// TIA Portal V21 export
FUNCTION "GestAzionamentoFesto_CMMT-ST" : Void   // FC43, LAD
{ S7_Optimized_Access := 'TRUE' }
// stored: SetENOAutomatically false
   VAR_INPUT
      "K_AzionamentoFesto_CMMT-ST" : Int;
      K_Motore : Int;
   END_VAR
   VAR_TEMP
      AzionamentoAbilitato : Bool;
      tempDWord : DWord;
      tmpSendBuffer : Array[0..11] of Word;
      tmpReadBuffer : Array[0..11] of Word;
      CambioPosPLC : Bool;
      CambioStatoMotore : Bool;
      ModePosDifferente : Bool;
      CambioStatoEnAxis : Bool;
      ResetRichiesto : Bool;
   END_VAR
   VAR CONSTANT
      MaxCounterStart : Int := 50;
      MAXMODE : Int := 8;
      STATUS_IN_OPERATION : Word := 16#7002;
      ERROR_INVALID_MODE : Word := 16#8202;
      ERROR_OVERRIDE : Word := 16#8203;
      ERROR_INVALID_TRV_BLOCK : Word := 16#8204;
      ERROR_DRIVE_ERROR : Word := 16#8401;
      ERROR_SWITCH_ON_INHIBITED : Word := 16#8402;
      ERROR_DPRD_DAT : Word := 16#8600;
      ERROR_DPWR_DAT : Word := 16#8601;
      Automode : Int := 2;
      JogMode : Int := 7;
      Homing : Int := 4;
   END_VAR
   VAR_TEMP   // added for the SCL form of the ladder/FBD networks
      _w1 : Bool;
   END_VAR
BEGIN

REGION Network 1
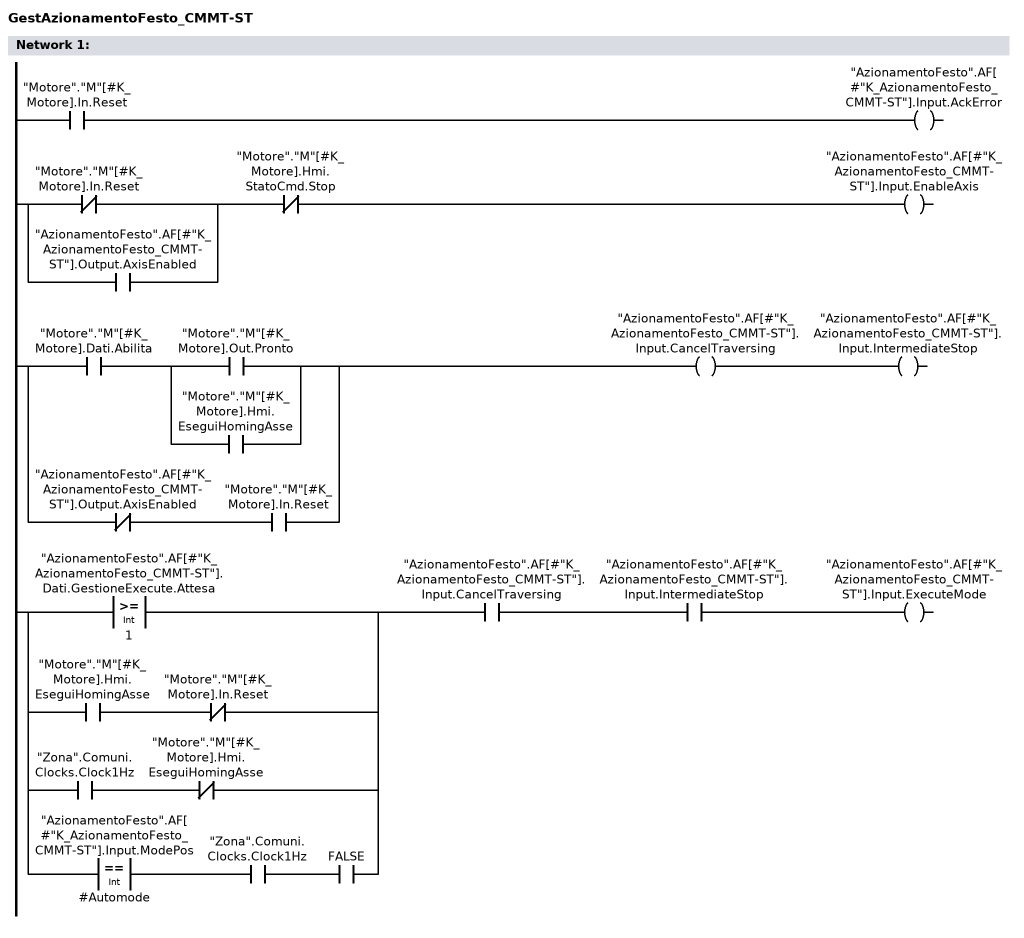
   RUNG wire#powerrail
      Contact( "Motore"."M"[#K_Motore].In.Reset )
      Coil( "AzionamentoFesto".AF[#"K_AzionamentoFesto_CMMT-ST"].Input.AckError )
   END_RUNG
   RUNG wire#powerrail
      I_Contact( "Motore"."M"[#K_Motore].In.Reset )
      wire#w1
      I_Contact( "Motore"."M"[#K_Motore].Hmi.StatoCmd.Stop )
      Coil( "AzionamentoFesto".AF[#"K_AzionamentoFesto_CMMT-ST"].Input.EnableAxis )
   END_RUNG
   RUNG wire#powerrail
      Contact( "AzionamentoFesto".AF[#"K_AzionamentoFesto_CMMT-ST"].Output.AxisEnabled )
   END_RUNG wire#w1
   RUNG wire#powerrail
      Contact( "Motore"."M"[#K_Motore].Dati.Abilita )
      wire#w2
      Contact( "Motore"."M"[#K_Motore].Out.Pronto )
      wire#w3
      Coil( "AzionamentoFesto".AF[#"K_AzionamentoFesto_CMMT-ST"].Input.CancelTraversing )
      Coil( "AzionamentoFesto".AF[#"K_AzionamentoFesto_CMMT-ST"].Input.IntermediateStop )
   END_RUNG
   RUNG wire#w2
      Contact( "Motore"."M"[#K_Motore].Hmi.EseguiHomingAsse )
   END_RUNG wire#w3
   RUNG wire#powerrail
      I_Contact( "AzionamentoFesto".AF[#"K_AzionamentoFesto_CMMT-ST"].Output.AxisEnabled )
      Contact( "Motore"."M"[#K_Motore].In.Reset )
   END_RUNG wire#w3
   RUNG wire#powerrail
      { S7_Templates := "SrcType := Int" } GE_Contact(in1 := "AzionamentoFesto".AF[#"K_AzionamentoFesto_CMMT-ST"].Dati.GestioneExecute.Attesa, in2 := 1)
      wire#w4
      Contact( "AzionamentoFesto".AF[#"K_AzionamentoFesto_CMMT-ST"].Input.CancelTraversing )
      Contact( "AzionamentoFesto".AF[#"K_AzionamentoFesto_CMMT-ST"].Input.IntermediateStop )
      Coil( "AzionamentoFesto".AF[#"K_AzionamentoFesto_CMMT-ST"].Input.ExecuteMode )
   END_RUNG
   RUNG wire#powerrail
      Contact( "Motore"."M"[#K_Motore].Hmi.EseguiHomingAsse )
      I_Contact( "Motore"."M"[#K_Motore].In.Reset )
   END_RUNG wire#w4
   RUNG wire#powerrail
      Contact( "Zona".Comuni.Clocks.Clock1Hz )
      I_Contact( "Motore"."M"[#K_Motore].Hmi.EseguiHomingAsse )
   END_RUNG wire#w4
   RUNG wire#powerrail
      { S7_Templates := "SrcType := Int" } EQ_Contact(in1 := "AzionamentoFesto".AF[#"K_AzionamentoFesto_CMMT-ST"].Input.ModePos, in2 := #Automode)
      Contact( "Zona".Comuni.Clocks.Clock1Hz )
      Contact( FALSE )
   END_RUNG wire#w4
   // the same network as SCL:
   "AzionamentoFesto".AF[#"K_AzionamentoFesto_CMMT-ST"].Input.AckError := "Motore"."M"[#K_Motore].In.Reset;
   "AzionamentoFesto".AF[#"K_AzionamentoFesto_CMMT-ST"].Input.EnableAxis := (NOT "Motore"."M"[#K_Motore].In.Reset OR "AzionamentoFesto".AF[#"K_AzionamentoFesto_CMMT-ST"].Output.AxisEnabled) AND NOT "Motore"."M"[#K_Motore].Hmi.StatoCmd.Stop;
   #_w1 := ("Motore"."M"[#K_Motore].Dati.Abilita AND ("Motore"."M"[#K_Motore].Out.Pronto OR "Motore"."M"[#K_Motore].Hmi.EseguiHomingAsse)) OR (NOT "AzionamentoFesto".AF[#"K_AzionamentoFesto_CMMT-ST"].Output.AxisEnabled AND "Motore"."M"[#K_Motore].In.Reset);
   "AzionamentoFesto".AF[#"K_AzionamentoFesto_CMMT-ST"].Input.CancelTraversing := #_w1;
   "AzionamentoFesto".AF[#"K_AzionamentoFesto_CMMT-ST"].Input.IntermediateStop := #_w1;
   "AzionamentoFesto".AF[#"K_AzionamentoFesto_CMMT-ST"].Input.ExecuteMode := (("AzionamentoFesto".AF[#"K_AzionamentoFesto_CMMT-ST"].Dati.GestioneExecute.Attesa >= 1) OR ("Motore"."M"[#K_Motore].Hmi.EseguiHomingAsse AND NOT "Motore"."M"[#K_Motore].In.Reset) OR ("Zona".Comuni.Clocks.Clock1Hz AND NOT "Motore"."M"[#K_Motore].Hmi.EseguiHomingAsse) OR (("AzionamentoFesto".AF[#"K_AzionamentoFesto_CMMT-ST"].Input.ModePos = #Automode) AND "Zona".Comuni.Clocks.Clock1Hz AND FALSE)) AND "AzionamentoFesto".AF[#"K_AzionamentoFesto_CMMT-ST"].Input.CancelTraversing AND "AzionamentoFesto".AF[#"K_AzionamentoFesto_CMMT-ST"].Input.IntermediateStop;
END_REGION

REGION Network 2 (SCL)
   REGION Modifiche from BRAIN ELECTRIC     

       "AzionamentoFesto".AF[#"K_AzionamentoFesto_CMMT-ST"].Input.HardwareId := "Motore".M[#K_Motore].In.ProfinetHwSubModule;
       "AzionamentoFesto".AF[#"K_AzionamentoFesto_CMMT-ST"].Input.Position := REAL_TO_DINT("Motore".M[#K_Motore].In.CmdPosizioneRich);
       "AzionamentoFesto".AF[#"K_AzionamentoFesto_CMMT-ST"].Input.Velocity := REAL_TO_INT("Motore".M[#K_Motore].In.CmdVelocitaRich);
       "AzionamentoFesto".AF[#"K_AzionamentoFesto_CMMT-ST"].Input.ConfigEPos := 15;



       REGION Comando execute nel motore

           IF "AzionamentoFesto".AF[#"K_AzionamentoFesto_CMMT-ST"].Dati.GestioneExecute.Richiesto AND "AzionamentoFesto".AF[#"K_AzionamentoFesto_CMMT-ST"].Dati.GestioneExecute.Attesa <= 5 THEN
               "AzionamentoFesto".AF[#"K_AzionamentoFesto_CMMT-ST"].Dati.GestioneExecute.Attesa += 1;
           END_IF;
           IF "AzionamentoFesto".AF[#"K_AzionamentoFesto_CMMT-ST"].Dati.GestioneExecute.Attesa >= 1 THEN
               "AzionamentoFesto".AF[#"K_AzionamentoFesto_CMMT-ST"].Dati.GestioneExecute.Durata += 1;
           END_IF;
           IF "AzionamentoFesto".AF[#"K_AzionamentoFesto_CMMT-ST"].Dati.GestioneExecute.Durata >= 2 OR "Motore".M[#K_Motore].Hmi.EseguiHomingAsse THEN
               "AzionamentoFesto".AF[#"K_AzionamentoFesto_CMMT-ST"].Dati.GestioneExecute.Richiesto := False;
               "AzionamentoFesto".AF[#"K_AzionamentoFesto_CMMT-ST"].Dati.GestioneExecute.Attesa :=
               "AzionamentoFesto".AF[#"K_AzionamentoFesto_CMMT-ST"].Dati.GestioneExecute.Durata := 0;
           END_IF;

               #CambioPosPLC := "AzionamentoFesto".AF[#"K_AzionamentoFesto_CMMT-ST"].Dati.GestioneExecute.OldPosition <> "AzionamentoFesto".AF[#"K_AzionamentoFesto_CMMT-ST"].Input.Position;
               #CambioStatoMotore := "AzionamentoFesto".AF[#"K_AzionamentoFesto_CMMT-ST"].Dati.GestioneExecute.OldStatoMotore <> "Motore".M[#K_Motore].Hmi.StatoMotore;
               #ModePosDifferente := "AzionamentoFesto".AF[#"K_AzionamentoFesto_CMMT-ST"].Input.ModePos <> "AzionamentoFesto".AF[#"K_AzionamentoFesto_CMMT-ST"].Dati.GestioneExecute.OldModePos;
               #CambioStatoEnAxis := "AzionamentoFesto".AF[#"K_AzionamentoFesto_CMMT-ST"].Input.EnableAxis <> "AzionamentoFesto".AF[#"K_AzionamentoFesto_CMMT-ST"].Dati.GestioneExecute.OldAxisEnable;
               #ResetRichiesto := "Motore".M[#K_Motore].In.Reset <> "AzionamentoFesto".AF[#"K_AzionamentoFesto_CMMT-ST"].Dati.GestioneExecute.OldResetState;
               IF #CambioPosPLC OR #CambioStatoMotore OR #ModePosDifferente OR #CambioStatoEnAxis OR #ResetRichiesto THEN
                   "AzionamentoFesto".AF[#"K_AzionamentoFesto_CMMT-ST"].Dati.GestioneExecute.OldPosition := "AzionamentoFesto".AF[#"K_AzionamentoFesto_CMMT-ST"].Input.Position;
                   "AzionamentoFesto".AF[#"K_AzionamentoFesto_CMMT-ST"].Dati.GestioneExecute.OldStatoMotore := "Motore".M[#K_Motore].Hmi.StatoMotore;
                   "AzionamentoFesto".AF[#"K_AzionamentoFesto_CMMT-ST"].Dati.GestioneExecute.OldAxisEnable := "AzionamentoFesto".AF[#"K_AzionamentoFesto_CMMT-ST"].Input.EnableAxis;
                   "AzionamentoFesto".AF[#"K_AzionamentoFesto_CMMT-ST"].Dati.GestioneExecute.OldModePos := "AzionamentoFesto".AF[#"K_AzionamentoFesto_CMMT-ST"].Input.ModePos;
                   "AzionamentoFesto".AF[#"K_AzionamentoFesto_CMMT-ST"].Dati.GestioneExecute.OldResetState := "Motore".M[#K_Motore].In.Reset;
                   "AzionamentoFesto".AF[#"K_AzionamentoFesto_CMMT-ST"].Dati.GestioneExecute.Richiesto := True;
               END_IF;
           END_REGION ;


       IF "Zona".Comuni.FirstScanFromCpu OR NOT "AzionamentoFesto".AF[#"K_AzionamentoFesto_CMMT-ST"].Output.AxisRef THEN
           "Motore".M[#K_Motore].Allarmi.A[KAllMot_RichiestaAzzeramento].Stato := True;
       END_IF;

       "Motore".M[#K_Motore].Out.PosAttuale := "AzionamentoFesto".AF[#"K_AzionamentoFesto_CMMT-ST"].Output.ActPosition;
       "Motore".M[#K_Motore].Allarmi.A[KAllMot_DriveInAllarme].Stato := "AzionamentoFesto".AF[#"K_AzionamentoFesto_CMMT-ST"].Output.AxisError;
       #AzionamentoAbilitato := "AzionamentoFesto".AF[#"K_AzionamentoFesto_CMMT-ST"].Output.AxisEnabled;

       IF NOT "Motore".M[#K_Motore].Hmi.EseguiHomingAsse THEN
           IF "Motore".M[#K_Motore].Hmi.StatoCmd.Stop OR NOT #AzionamentoAbilitato THEN
               "AzionamentoFesto".AF[#"K_AzionamentoFesto_CMMT-ST"].Input.ModePos := #Automode;
               "AzionamentoFesto".AF[#"K_AzionamentoFesto_CMMT-ST"].Input.Jog1 := False;
               "AzionamentoFesto".AF[#"K_AzionamentoFesto_CMMT-ST"].Input.Jog2 := False;
               "AzionamentoFesto".AF[#"K_AzionamentoFesto_CMMT-ST"].Input.OverV := 0;
               "AzionamentoFesto".AF[#"K_AzionamentoFesto_CMMT-ST"].Input.Velocity := 0;
           ELSIF "Motore".M[#K_Motore].Hmi.StatoCmd.Auto THEN
               "AzionamentoFesto".AF[#"K_AzionamentoFesto_CMMT-ST"].Input.ModePos := #Automode;
               "AzionamentoFesto".AF[#"K_AzionamentoFesto_CMMT-ST"].Input.Jog1 := False;
               "AzionamentoFesto".AF[#"K_AzionamentoFesto_CMMT-ST"].Input.Jog2 := False;
               "AzionamentoFesto".AF[#"K_AzionamentoFesto_CMMT-ST"].Input.OverV := 100;
           ELSIF "Motore".M[#K_Motore].Hmi.StatoCmd.ManPos THEN
               "AzionamentoFesto".AF[#"K_AzionamentoFesto_CMMT-ST"].Input.ModePos := #JogMode;
               "AzionamentoFesto".AF[#"K_AzionamentoFesto_CMMT-ST"].Input.Jog1 := True;
               "AzionamentoFesto".AF[#"K_AzionamentoFesto_CMMT-ST"].Input.OverV := REAL_TO_INT("Motore".M[#K_Motore].Hmi.VelManuale);
           ELSIF "Motore".M[#K_Motore].Hmi.StatoCmd.ManNeg THEN
               "AzionamentoFesto".AF[#"K_AzionamentoFesto_CMMT-ST"].Input.ModePos := #JogMode;
               "AzionamentoFesto".AF[#"K_AzionamentoFesto_CMMT-ST"].Input.Jog2 := True;
               "AzionamentoFesto".AF[#"K_AzionamentoFesto_CMMT-ST"].Input.OverV := REAL_TO_INT("Motore".M[#K_Motore].Hmi.VelManuale);
           END_IF;
       ELSE
           "AzionamentoFesto".AF[#"K_AzionamentoFesto_CMMT-ST"].Input.ModePos := #Homing;
           "AzionamentoFesto".AF[#"K_AzionamentoFesto_CMMT-ST"].Input.Jog1 := False;
           "AzionamentoFesto".AF[#"K_AzionamentoFesto_CMMT-ST"].Input.Jog2 := False;
           "AzionamentoFesto".AF[#"K_AzionamentoFesto_CMMT-ST"].Input.OverV := REAL_TO_INT("Motore".M[#K_Motore].Hmi.VelManuale);
           "AzionamentoFesto".AF[#"K_AzionamentoFesto_CMMT-ST"].Input.Velocity := 100;
       END_IF;
       IF "AzionamentoFesto".AF[#"K_AzionamentoFesto_CMMT-ST"].Output.AxisRef AND "Motore".M[#K_Motore].Hmi.EseguiHomingAsse THEN //OR NOT "AzionamentiFesto".AF[#"K_AzionamentoFesto_CMMT-ST"].Input.EnableAxis THEN
           "Motore".M[#K_Motore].Hmi.EseguiHomingAsse := False;
           "Motore".M[#K_Motore].Allarmi.A[KAllMot_RichiestaAzzeramento].Stato := False;
       END_IF;

   END_REGION
   REGION Check OPM and Override Values
       // Check the Mode of Operation
       IF "AzionamentoFesto".AF[#"K_AzionamentoFesto_CMMT-ST"].Input.ModePos > #MAXMODE THEN
           "AzionamentoFesto".AF[#"K_AzionamentoFesto_CMMT-ST"].Output.Error := True;
           "AzionamentoFesto".AF[#"K_AzionamentoFesto_CMMT-ST"].Dati.Status := #ERROR_INVALID_MODE;
           "AzionamentoFesto".AF[#"K_AzionamentoFesto_CMMT-ST"].Dati.ExecuteIntern := false;
       ELSIF "AzionamentoFesto".AF[#"K_AzionamentoFesto_CMMT-ST"].Input.ModePos < 1 THEN
           "AzionamentoFesto".AF[#"K_AzionamentoFesto_CMMT-ST"].Output.Error := True;
           "AzionamentoFesto".AF[#"K_AzionamentoFesto_CMMT-ST"].Dati.Status := #ERROR_INVALID_MODE;
           "AzionamentoFesto".AF[#"K_AzionamentoFesto_CMMT-ST"].Dati.ExecuteIntern := false;
       ELSE
           IF "AzionamentoFesto".AF[#"K_AzionamentoFesto_CMMT-ST"].Dati.Status = #ERROR_INVALID_MODE THEN
               "AzionamentoFesto".AF[#"K_AzionamentoFesto_CMMT-ST"].Dati.Status := #STATUS_IN_OPERATION;
               "AzionamentoFesto".AF[#"K_AzionamentoFesto_CMMT-ST"].Output.Error := False;
           END_IF;
       END_IF;


       //Check the Velocity Override 
       IF ("AzionamentoFesto".AF[#"K_AzionamentoFesto_CMMT-ST"].Input.OverV < 0) OR ("AzionamentoFesto".AF[#"K_AzionamentoFesto_CMMT-ST"].Input.OverV > 199) THEN
           "AzionamentoFesto".AF[#"K_AzionamentoFesto_CMMT-ST"].Dati.Status := #ERROR_OVERRIDE;
           "AzionamentoFesto".AF[#"K_AzionamentoFesto_CMMT-ST"].Output.Error := True;
       ELSE
           // Write Velocity Override into Send Buffer
           "AzionamentoFesto".AF[#"K_AzionamentoFesto_CMMT-ST"].Dati.CycWrite.Override := INT_TO_WORD(REAL_TO_INT(16384.0 * (INT_TO_REAL("AzionamentoFesto".AF[#"K_AzionamentoFesto_CMMT-ST"].Input.OverV) / 100.0)));
           IF "AzionamentoFesto".AF[#"K_AzionamentoFesto_CMMT-ST"].Dati.Status = #ERROR_OVERRIDE THEN
               "AzionamentoFesto".AF[#"K_AzionamentoFesto_CMMT-ST"].Dati.Status := #STATUS_IN_OPERATION;
               "AzionamentoFesto".AF[#"K_AzionamentoFesto_CMMT-ST"].Output.Error := False;
           END_IF;
       END_IF;

       //Check the Acceleration Override  (0% - 100%, 100% => W#16#4000)
       IF ("AzionamentoFesto".AF[#"K_AzionamentoFesto_CMMT-ST"].Input.OverAcc < 0) OR ("AzionamentoFesto".AF[#"K_AzionamentoFesto_CMMT-ST"].Input.OverAcc > 100) THEN
           "AzionamentoFesto".AF[#"K_AzionamentoFesto_CMMT-ST"].Dati.Status := #ERROR_OVERRIDE;
           "AzionamentoFesto".AF[#"K_AzionamentoFesto_CMMT-ST"].Output.Error := True;
       ELSE
           // Write Acceleration Override into Send Buffer
           "AzionamentoFesto".AF[#"K_AzionamentoFesto_CMMT-ST"].Dati.CycWrite.MDI_ACC := INT_TO_WORD(REAL_TO_INT(16384.0 * (INT_TO_REAL("AzionamentoFesto".AF[#"K_AzionamentoFesto_CMMT-ST"].Input.OverAcc) / 100.0)));
           IF "AzionamentoFesto".AF[#"K_AzionamentoFesto_CMMT-ST"].Dati.Status = #ERROR_OVERRIDE THEN
               "AzionamentoFesto".AF[#"K_AzionamentoFesto_CMMT-ST"].Dati.Status := #STATUS_IN_OPERATION;
               "AzionamentoFesto".AF[#"K_AzionamentoFesto_CMMT-ST"].Output.Error := False;
           END_IF;
       END_IF;

       //Check the Deceleration Override  (0% - 100%, 100% => W#16#4000)
       IF ("AzionamentoFesto".AF[#"K_AzionamentoFesto_CMMT-ST"].Input.OverDec < 0) OR ("AzionamentoFesto".AF[#"K_AzionamentoFesto_CMMT-ST"].Input.OverDec > 100) THEN
           "AzionamentoFesto".AF[#"K_AzionamentoFesto_CMMT-ST"].Dati.Status := #ERROR_OVERRIDE;
           "AzionamentoFesto".AF[#"K_AzionamentoFesto_CMMT-ST"].Output.Error := True;
       ELSE
           // Write Deceleration Override into Send Buffer
           "AzionamentoFesto".AF[#"K_AzionamentoFesto_CMMT-ST"].Dati.CycWrite.MDI_DEC := INT_TO_WORD(REAL_TO_INT(16384.0 * (INT_TO_REAL("AzionamentoFesto".AF[#"K_AzionamentoFesto_CMMT-ST"].Input.OverDec) / 100.0)));
           IF "AzionamentoFesto".AF[#"K_AzionamentoFesto_CMMT-ST"].Dati.Status = #ERROR_OVERRIDE THEN
               "AzionamentoFesto".AF[#"K_AzionamentoFesto_CMMT-ST"].Dati.Status := #STATUS_IN_OPERATION;
               "AzionamentoFesto".AF[#"K_AzionamentoFesto_CMMT-ST"].Output.Error := False;
           END_IF;
       END_IF;
   END_REGION ;

   REGION Lettura della status word
       // Read cyclic telegram 111
       "AzionamentoFesto".AF[#"K_AzionamentoFesto_CMMT-ST"].Dati.RetDPRD := DPRD_DAT(LADDR := "AzionamentoFesto".AF[#"K_AzionamentoFesto_CMMT-ST"].Input.HardwareId,
                                                                                     RECORD => #tmpReadBuffer);

       //check if the return code is unequal zero -> error occured
       IF "AzionamentoFesto".AF[#"K_AzionamentoFesto_CMMT-ST"].Dati.RetDPRD <> 0 THEN
           "AzionamentoFesto".AF[#"K_AzionamentoFesto_CMMT-ST"].Output.Error := true;
           "AzionamentoFesto".AF[#"K_AzionamentoFesto_CMMT-ST"].Dati.Status := #ERROR_DPRD_DAT;
           "AzionamentoFesto".AF[#"K_AzionamentoFesto_CMMT-ST"].Output.DiagID := INT_TO_WORD("AzionamentoFesto".AF[#"K_AzionamentoFesto_CMMT-ST"].Dati.RetDPRD);
       ELSE

           // set the Diag status back "in operation"
           IF "AzionamentoFesto".AF[#"K_AzionamentoFesto_CMMT-ST"].Dati.Status = #ERROR_DPRD_DAT THEN
               "AzionamentoFesto".AF[#"K_AzionamentoFesto_CMMT-ST"].Dati.Status := #STATUS_IN_OPERATION;
               "AzionamentoFesto".AF[#"K_AzionamentoFesto_CMMT-ST"].Output.DiagID := 0;
               "AzionamentoFesto".AF[#"K_AzionamentoFesto_CMMT-ST"].Output.Error := False;
           END_IF;
       END_IF;

   END_REGION ;


   REGION Read Input from temp data
       // copy all values from tmp buffer to static data
       // ZSW1
       "AzionamentoFesto".AF[#"K_AzionamentoFesto_CMMT-ST"].Dati.CycRead.ZSW1.followingErrorInTolerance := #tmpReadBuffer[0].%X8;
       "AzionamentoFesto".AF[#"K_AzionamentoFesto_CMMT-ST"].Dati.CycRead.ZSW1.controlRequest := #tmpReadBuffer[0].%X9;
       "AzionamentoFesto".AF[#"K_AzionamentoFesto_CMMT-ST"].Dati.CycRead.ZSW1.targetPosReached := #tmpReadBuffer[0].%X10;
       "AzionamentoFesto".AF[#"K_AzionamentoFesto_CMMT-ST"].Dati.CycRead.ZSW1.homePosSet := #tmpReadBuffer[0].%X11;
       "AzionamentoFesto".AF[#"K_AzionamentoFesto_CMMT-ST"].Dati.CycRead.ZSW1.acknowledgeTraversingBlockActivated := #tmpReadBuffer[0].%X12;
       "AzionamentoFesto".AF[#"K_AzionamentoFesto_CMMT-ST"].Dati.CycRead.ZSW1.driveStopped := #tmpReadBuffer[0].%X13;
       "AzionamentoFesto".AF[#"K_AzionamentoFesto_CMMT-ST"].Dati.CycRead.ZSW1.axisAccelerates := #tmpReadBuffer[0].%X14;
       "AzionamentoFesto".AF[#"K_AzionamentoFesto_CMMT-ST"].Dati.CycRead.ZSW1.axisDecelerates := #tmpReadBuffer[0].%X15;
       "AzionamentoFesto".AF[#"K_AzionamentoFesto_CMMT-ST"].Dati.CycRead.ZSW1.readyForSwitchOn := #tmpReadBuffer[0].%X0;
       "AzionamentoFesto".AF[#"K_AzionamentoFesto_CMMT-ST"].Dati.CycRead.ZSW1.ready := #tmpReadBuffer[0].%X1;
       "AzionamentoFesto".AF[#"K_AzionamentoFesto_CMMT-ST"].Dati.CycRead.ZSW1.operationEnabled := #tmpReadBuffer[0].%X2;
       "AzionamentoFesto".AF[#"K_AzionamentoFesto_CMMT-ST"].Dati.CycRead.ZSW1.faultPresent := #tmpReadBuffer[0].%X3;
       "AzionamentoFesto".AF[#"K_AzionamentoFesto_CMMT-ST"].Dati.CycRead.ZSW1.noCoastingActive := #tmpReadBuffer[0].%X4;
       "AzionamentoFesto".AF[#"K_AzionamentoFesto_CMMT-ST"].Dati.CycRead.ZSW1.noQuickStopActive := #tmpReadBuffer[0].%X5;
       "AzionamentoFesto".AF[#"K_AzionamentoFesto_CMMT-ST"].Dati.CycRead.ZSW1.switchingOnInhibitedActive := #tmpReadBuffer[0].%X6;
       "AzionamentoFesto".AF[#"K_AzionamentoFesto_CMMT-ST"].Dati.CycRead.ZSW1.warningActive := #tmpReadBuffer[0].%X7;

       //POS_ZSW1
       "AzionamentoFesto".AF[#"K_AzionamentoFesto_CMMT-ST"].Dati.CycRead.POS_ZSW1 := #tmpReadBuffer[1];
       "AzionamentoFesto".AF[#"K_AzionamentoFesto_CMMT-ST"].Output.EPosZSW1 := "AzionamentoFesto".AF[#"K_AzionamentoFesto_CMMT-ST"].Dati.CycRead.POS_ZSW1;

       //POS_ZSW2
       "AzionamentoFesto".AF[#"K_AzionamentoFesto_CMMT-ST"].Dati.CycRead.POS_ZSW2 := #tmpReadBuffer[2];
       "AzionamentoFesto".AF[#"K_AzionamentoFesto_CMMT-ST"].Output.EPosZSW2 := "AzionamentoFesto".AF[#"K_AzionamentoFesto_CMMT-ST"].Dati.CycRead.POS_ZSW2;

       // ZSW2
       "AzionamentoFesto".AF[#"K_AzionamentoFesto_CMMT-ST"].Dati.CycRead.ZSW2.deviceSpecificBit8 := #tmpReadBuffer[3].%X8;
       "AzionamentoFesto".AF[#"K_AzionamentoFesto_CMMT-ST"].Dati.CycRead.ZSW2.deviceSpecificBit9 := #tmpReadBuffer[3].%X9;
       "AzionamentoFesto".AF[#"K_AzionamentoFesto_CMMT-ST"].Dati.CycRead.ZSW2.deviceSpecificBit10 := #tmpReadBuffer[3].%X10;
       "AzionamentoFesto".AF[#"K_AzionamentoFesto_CMMT-ST"].Dati.CycRead.ZSW2.deviceSpecificBit11 := #tmpReadBuffer[3].%X11;
       "AzionamentoFesto".AF[#"K_AzionamentoFesto_CMMT-ST"].Dati.CycRead.ZSW2.doSignOfLifeBit0 := #tmpReadBuffer[3].%X12;
       "AzionamentoFesto".AF[#"K_AzionamentoFesto_CMMT-ST"].Dati.CycRead.ZSW2.doSignOfLifeBit1 := #tmpReadBuffer[3].%X13;
       "AzionamentoFesto".AF[#"K_AzionamentoFesto_CMMT-ST"].Dati.CycRead.ZSW2.doSignOfLifeBit2 := #tmpReadBuffer[3].%X14;
       "AzionamentoFesto".AF[#"K_AzionamentoFesto_CMMT-ST"].Dati.CycRead.ZSW2.doSignOfLifeBit3 := #tmpReadBuffer[3].%X15;
       "AzionamentoFesto".AF[#"K_AzionamentoFesto_CMMT-ST"].Dati.CycRead.ZSW2.deviceSpecificBit0 := #tmpReadBuffer[3].%X0;
       "AzionamentoFesto".AF[#"K_AzionamentoFesto_CMMT-ST"].Dati.CycRead.ZSW2.deviceSpecificBit1 := #tmpReadBuffer[3].%X1;
       "AzionamentoFesto".AF[#"K_AzionamentoFesto_CMMT-ST"].Dati.CycRead.ZSW2.deviceSpecificBit2 := #tmpReadBuffer[3].%X2;
       "AzionamentoFesto".AF[#"K_AzionamentoFesto_CMMT-ST"].Dati.CycRead.ZSW2.deviceSpecificBit3 := #tmpReadBuffer[3].%X3;
       "AzionamentoFesto".AF[#"K_AzionamentoFesto_CMMT-ST"].Dati.CycRead.ZSW2.deviceSpecificBit4 := #tmpReadBuffer[3].%X4;
       "AzionamentoFesto".AF[#"K_AzionamentoFesto_CMMT-ST"].Dati.CycRead.ZSW2.deviceSpecificBit5 := #tmpReadBuffer[3].%X5;
       "AzionamentoFesto".AF[#"K_AzionamentoFesto_CMMT-ST"].Dati.CycRead.ZSW2.deviceSpecificBit6 := #tmpReadBuffer[3].%X6;
       "AzionamentoFesto".AF[#"K_AzionamentoFesto_CMMT-ST"].Dati.CycRead.ZSW2.deviceSpecificBit7 := #tmpReadBuffer[3].%X7;

       //MELDW
       "AzionamentoFesto".AF[#"K_AzionamentoFesto_CMMT-ST"].Dati.CycRead.MELDW := #tmpReadBuffer[4];

       //XIST_A
       "AzionamentoFesto".AF[#"K_AzionamentoFesto_CMMT-ST"].Dati.CycRead.XIST_A.%W0 := #tmpReadBuffer[6];
       "AzionamentoFesto".AF[#"K_AzionamentoFesto_CMMT-ST"].Dati.CycRead.XIST_A.%W1 := #tmpReadBuffer[5];

       //NIST_B
       "AzionamentoFesto".AF[#"K_AzionamentoFesto_CMMT-ST"].Dati.CycRead.NIST_B.%W0 := #tmpReadBuffer[8];
       "AzionamentoFesto".AF[#"K_AzionamentoFesto_CMMT-ST"].Dati.CycRead.NIST_B.%W1 := #tmpReadBuffer[7];

       //Fault_Code
       "AzionamentoFesto".AF[#"K_AzionamentoFesto_CMMT-ST"].Dati.CycRead.Fault_Code := #tmpReadBuffer[9];

       //Warn_Code
       "AzionamentoFesto".AF[#"K_AzionamentoFesto_CMMT-ST"].Dati.CycRead.Warn_Code := #tmpReadBuffer[10];

       //Reserved
       "AzionamentoFesto".AF[#"K_AzionamentoFesto_CMMT-ST"].Dati.CycRead.Reserved := #tmpReadBuffer[11];
   END_REGION ;

   // Mapping of the FB Outputs
   "AzionamentoFesto".AF[#"K_AzionamentoFesto_CMMT-ST"].Output.AxisEnabled := "AzionamentoFesto".AF[#"K_AzionamentoFesto_CMMT-ST"].Dati.CycRead.ZSW1.operationEnabled;
   "AzionamentoFesto".AF[#"K_AzionamentoFesto_CMMT-ST"].Output.AxisError := "AzionamentoFesto".AF[#"K_AzionamentoFesto_CMMT-ST"].Dati.CycRead.ZSW1.faultPresent;
   "AzionamentoFesto".AF[#"K_AzionamentoFesto_CMMT-ST"].Output.AxisWarn := "AzionamentoFesto".AF[#"K_AzionamentoFesto_CMMT-ST"].Dati.CycRead.ZSW1.warningActive;
   "AzionamentoFesto".AF[#"K_AzionamentoFesto_CMMT-ST"].Output.AxisPosOk := "AzionamentoFesto".AF[#"K_AzionamentoFesto_CMMT-ST"].Dati.CycRead.ZSW1.targetPosReached;
   "AzionamentoFesto".AF[#"K_AzionamentoFesto_CMMT-ST"].Output.AxisRef := "AzionamentoFesto".AF[#"K_AzionamentoFesto_CMMT-ST"].Dati.CycRead.ZSW1.homePosSet;
   "AzionamentoFesto".AF[#"K_AzionamentoFesto_CMMT-ST"].Output.AxisAckSetpoint := "AzionamentoFesto".AF[#"K_AzionamentoFesto_CMMT-ST"].Dati.CycRead.ZSW1.acknowledgeTraversingBlockActivated;
   "AzionamentoFesto".AF[#"K_AzionamentoFesto_CMMT-ST"].Output.ClampTorqueReached := "AzionamentoFesto".AF[#"K_AzionamentoFesto_CMMT-ST"].Dati.CycRead.POS_ZSW2.%X13;
   "AzionamentoFesto".AF[#"K_AzionamentoFesto_CMMT-ST"].Output.AxisSpFixed := "AzionamentoFesto".AF[#"K_AzionamentoFesto_CMMT-ST"].Dati.CycRead.ZSW1.driveStopped;
   "AzionamentoFesto".AF[#"K_AzionamentoFesto_CMMT-ST"].Output.ActVelocity := "AzionamentoFesto".AF[#"K_AzionamentoFesto_CMMT-ST"].Dati.CycRead.NIST_B;


   //scaling the ActVelocity output
   IF "AzionamentoFesto".AF[#"K_AzionamentoFesto_CMMT-ST"].Input.BaseSpeedValue <> 0 THEN
       "AzionamentoFesto".AF[#"K_AzionamentoFesto_CMMT-ST"].Output.ActVelocity := "AzionamentoFesto".AF[#"K_AzionamentoFesto_CMMT-ST"].Output.ActVelocity * (("AzionamentoFesto".AF[#"K_AzionamentoFesto_CMMT-ST"].Input.BaseSpeedValue / 1073741824.0));
   END_IF;

   "AzionamentoFesto".AF[#"K_AzionamentoFesto_CMMT-ST"].Output.ActPosition := "AzionamentoFesto".AF[#"K_AzionamentoFesto_CMMT-ST"].Dati.CycRead.XIST_A;
   "AzionamentoFesto".AF[#"K_AzionamentoFesto_CMMT-ST"].Output.ActWarn := "AzionamentoFesto".AF[#"K_AzionamentoFesto_CMMT-ST"].Dati.CycRead.Warn_Code;
   "AzionamentoFesto".AF[#"K_AzionamentoFesto_CMMT-ST"].Output.ActFault := "AzionamentoFesto".AF[#"K_AzionamentoFesto_CMMT-ST"].Dati.CycRead.Fault_Code;
   "AzionamentoFesto".AF[#"K_AzionamentoFesto_CMMT-ST"].Output.Lockout := "AzionamentoFesto".AF[#"K_AzionamentoFesto_CMMT-ST"].Dati.CycRead.ZSW1.switchingOnInhibitedActive;

   //Check the drive error and Lockout status
   IF "AzionamentoFesto".AF[#"K_AzionamentoFesto_CMMT-ST"].Output.AxisError THEN
       "AzionamentoFesto".AF[#"K_AzionamentoFesto_CMMT-ST"].Dati.Status := #ERROR_DRIVE_ERROR;
       "AzionamentoFesto".AF[#"K_AzionamentoFesto_CMMT-ST"].Output.Error := True;
   ELSIF "AzionamentoFesto".AF[#"K_AzionamentoFesto_CMMT-ST"].Output.Lockout THEN
       "AzionamentoFesto".AF[#"K_AzionamentoFesto_CMMT-ST"].Dati.Status := #ERROR_SWITCH_ON_INHIBITED;
       "AzionamentoFesto".AF[#"K_AzionamentoFesto_CMMT-ST"].Output.Error := True;
   ELSE
       // error is gone -> set status in operational
       IF ("AzionamentoFesto".AF[#"K_AzionamentoFesto_CMMT-ST"].Dati.Status = #ERROR_DRIVE_ERROR) OR "AzionamentoFesto".AF[#"K_AzionamentoFesto_CMMT-ST"].Dati.Status = #ERROR_SWITCH_ON_INHIBITED THEN
           "AzionamentoFesto".AF[#"K_AzionamentoFesto_CMMT-ST"].Dati.Status := #STATUS_IN_OPERATION;
           "AzionamentoFesto".AF[#"K_AzionamentoFesto_CMMT-ST"].Output.Error := False;
       END_IF;
   END_IF;

   //Enable the Axis
   "AzionamentoFesto".AF[#"K_AzionamentoFesto_CMMT-ST"].Dati.CycWrite.STW1.on := "AzionamentoFesto".AF[#"K_AzionamentoFesto_CMMT-ST"].Input.EnableAxis;                       //STW1.0

   //fix values for STW1 data
   "AzionamentoFesto".AF[#"K_AzionamentoFesto_CMMT-ST"].Dati.CycWrite.STW1.cancelTraversing := "AzionamentoFesto".AF[#"K_AzionamentoFesto_CMMT-ST"].Input.CancelTraversing;   //STW1.4
   "AzionamentoFesto".AF[#"K_AzionamentoFesto_CMMT-ST"].Dati.CycWrite.STW1.intermediateStop := "AzionamentoFesto".AF[#"K_AzionamentoFesto_CMMT-ST"].Input.IntermediateStop;   //STW1.5
   "AzionamentoFesto".AF[#"K_AzionamentoFesto_CMMT-ST"].Dati.CycWrite.STW1.acknowledgeFault := "AzionamentoFesto".AF[#"K_AzionamentoFesto_CMMT-ST"].Input.AckError;           //STW1.7
   "AzionamentoFesto".AF[#"K_AzionamentoFesto_CMMT-ST"].Dati.CycWrite.STW1.controlByPlc := TRUE;                    //STW1.10
   "AzionamentoFesto".AF[#"K_AzionamentoFesto_CMMT-ST"].Dati.CycWrite.STW1.enableOperation := TRUE;                 //STW1.3

   // copy the position set value into the send struct
   IF "AzionamentoFesto".AF[#"K_AzionamentoFesto_CMMT-ST"].Input.ModePos <> 4 OR "AzionamentoFesto".AF[#"K_AzionamentoFesto_CMMT-ST"].Input.ModePos <> 5 OR "AzionamentoFesto".AF[#"K_AzionamentoFesto_CMMT-ST"].Input.ModePos <> 6 OR "AzionamentoFesto".AF[#"K_AzionamentoFesto_CMMT-ST"].Input.ModePos <> 7 OR "AzionamentoFesto".AF[#"K_AzionamentoFesto_CMMT-ST"].Input.ModePos <> 8 THEN
       "AzionamentoFesto".AF[#"K_AzionamentoFesto_CMMT-ST"].Dati.CycWrite.MDI_TARPOS := "AzionamentoFesto".AF[#"K_AzionamentoFesto_CMMT-ST"].Input.Position;
   ELSE
       "AzionamentoFesto".AF[#"K_AzionamentoFesto_CMMT-ST"].Dati.CycWrite.MDI_TARPOS := 0;
   END_IF;

   //copy the velocity set value into the send struct
   "AzionamentoFesto".AF[#"K_AzionamentoFesto_CMMT-ST"].Dati.CycWrite.MDI_VELOCITY := "AzionamentoFesto".AF[#"K_AzionamentoFesto_CMMT-ST"].Input.Velocity;

   //Jog bits
   // Mode 7
   //Generate the Jog1 Edge
   "AzionamentoFesto".AF[#"K_AzionamentoFesto_CMMT-ST"].Dati.Jog1PR_trig := "AzionamentoFesto".AF[#"K_AzionamentoFesto_CMMT-ST"].Input.Jog1 AND NOT "AzionamentoFesto".AF[#"K_AzionamentoFesto_CMMT-ST"].Dati.Jog1PAux;
   //Reset the Auxiliary flag 
   "AzionamentoFesto".AF[#"K_AzionamentoFesto_CMMT-ST"].Dati.Jog1PAux := "AzionamentoFesto".AF[#"K_AzionamentoFesto_CMMT-ST"].Input.Jog1;

   //Generate the Jog2 Edge
   "AzionamentoFesto".AF[#"K_AzionamentoFesto_CMMT-ST"].Dati.Jog2PR_trig := "AzionamentoFesto".AF[#"K_AzionamentoFesto_CMMT-ST"].Input.Jog2 AND NOT "AzionamentoFesto".AF[#"K_AzionamentoFesto_CMMT-ST"].Dati.Jog2PAux;
   //Reset the Auxiliary flag 
   "AzionamentoFesto".AF[#"K_AzionamentoFesto_CMMT-ST"].Dati.Jog2PAux := "AzionamentoFesto".AF[#"K_AzionamentoFesto_CMMT-ST"].Input.Jog2;

   //Mode 8
   //Generate the Jog1 Edge
   "AzionamentoFesto".AF[#"K_AzionamentoFesto_CMMT-ST"].Dati.Jog1PMode8R_trig := "AzionamentoFesto".AF[#"K_AzionamentoFesto_CMMT-ST"].Input.Jog1 AND NOT "AzionamentoFesto".AF[#"K_AzionamentoFesto_CMMT-ST"].Dati.Jog1PMode8Aux;
   //Reset the Auxiliary flag 
   "AzionamentoFesto".AF[#"K_AzionamentoFesto_CMMT-ST"].Dati.Jog1PMode8Aux := "AzionamentoFesto".AF[#"K_AzionamentoFesto_CMMT-ST"].Input.Jog1;

   //Generate the Jog2 Edge
   "AzionamentoFesto".AF[#"K_AzionamentoFesto_CMMT-ST"].Dati.Jog2PMode8R_trig := "AzionamentoFesto".AF[#"K_AzionamentoFesto_CMMT-ST"].Input.Jog2 AND NOT "AzionamentoFesto".AF[#"K_AzionamentoFesto_CMMT-ST"].Dati.Jog2PMode8Aux;
   //Reset the Auxiliary flag 
   "AzionamentoFesto".AF[#"K_AzionamentoFesto_CMMT-ST"].Dati.Jog2PMode8Aux := "AzionamentoFesto".AF[#"K_AzionamentoFesto_CMMT-ST"].Input.Jog2;

   IF "AzionamentoFesto".AF[#"K_AzionamentoFesto_CMMT-ST"].Input.ModePos <> 4 THEN
       //Start homing
       "AzionamentoFesto".AF[#"K_AzionamentoFesto_CMMT-ST"].Dati.CycWrite.STW1.StartHoming := false;
   END_IF;

   //Relative - Absolute
   "AzionamentoFesto".AF[#"K_AzionamentoFesto_CMMT-ST"].Dati.CycWrite.POS_STW1.MDI_MOD := false;

   //Positive - Negative direction
   "AzionamentoFesto".AF[#"K_AzionamentoFesto_CMMT-ST"].Dati.CycWrite.POS_STW1.PosModulo := false;
   "AzionamentoFesto".AF[#"K_AzionamentoFesto_CMMT-ST"].Dati.CycWrite.POS_STW1.NegModulo := false;

   // setup mode 
   "AzionamentoFesto".AF[#"K_AzionamentoFesto_CMMT-ST"].Dati.CycWrite.POS_STW1.SetupMode := false;

   // MDI Active
   "AzionamentoFesto".AF[#"K_AzionamentoFesto_CMMT-ST"].Dati.CycWrite.POS_STW1.MDI_Activate := false;

   //Trackingmode
   "AzionamentoFesto".AF[#"K_AzionamentoFesto_CMMT-ST"].Dati.CycWrite.POS_STW2.Trackingmode := false;

   //Jog increment
   "AzionamentoFesto".AF[#"K_AzionamentoFesto_CMMT-ST"].Dati.CycWrite.POS_STW2.jog_inc := false;

   //delete all the record bits
   "AzionamentoFesto".AF[#"K_AzionamentoFesto_CMMT-ST"].Dati.CycWrite.POS_STW1.travBlockBit0 := false;
   "AzionamentoFesto".AF[#"K_AzionamentoFesto_CMMT-ST"].Dati.CycWrite.POS_STW1.travBlockBit1 := false;
   "AzionamentoFesto".AF[#"K_AzionamentoFesto_CMMT-ST"].Dati.CycWrite.POS_STW1.travBlockBit2 := false;
   "AzionamentoFesto".AF[#"K_AzionamentoFesto_CMMT-ST"].Dati.CycWrite.POS_STW1.travBlockBit3 := false;
   "AzionamentoFesto".AF[#"K_AzionamentoFesto_CMMT-ST"].Dati.CycWrite.POS_STW1.travBlockBit4 := false;
   "AzionamentoFesto".AF[#"K_AzionamentoFesto_CMMT-ST"].Dati.CycWrite.POS_STW1.travBlockBit5 := false;
   "AzionamentoFesto".AF[#"K_AzionamentoFesto_CMMT-ST"].Dati.CycWrite.POS_STW1.travBlockBit6 := false;

   //Check if the drive is ready for a motion
   IF "AzionamentoFesto".AF[#"K_AzionamentoFesto_CMMT-ST"].Dati.CycRead.ZSW1.operationEnabled THEN
       "AzionamentoFesto".AF[#"K_AzionamentoFesto_CMMT-ST"].Dati.Ready4Motion := true;
   ELSE
       "AzionamentoFesto".AF[#"K_AzionamentoFesto_CMMT-ST"].Dati.Ready4Motion := false;
   END_IF;

   //Generate the Execute Edge for Mode = 4 and 5
   "AzionamentoFesto".AF[#"K_AzionamentoFesto_CMMT-ST"].Dati.ExecR_Trig := "AzionamentoFesto".AF[#"K_AzionamentoFesto_CMMT-ST"].Input.ExecuteMode AND NOT "AzionamentoFesto".AF[#"K_AzionamentoFesto_CMMT-ST"].Dati.ExecAux;
   //Reset the Auxiliary flag 
   "AzionamentoFesto".AF[#"K_AzionamentoFesto_CMMT-ST"].Dati.ExecAux := "AzionamentoFesto".AF[#"K_AzionamentoFesto_CMMT-ST"].Input.ExecuteMode;

   // Set the Execute command according to the ModePos
   IF NOT "AzionamentoFesto".AF[#"K_AzionamentoFesto_CMMT-ST"].Input.ExecuteMode THEN
       "AzionamentoFesto".AF[#"K_AzionamentoFesto_CMMT-ST"].Dati.ExecuteIntern := FALSE;
       "AzionamentoFesto".AF[#"K_AzionamentoFesto_CMMT-ST"].Dati.StepHome := 0;
   ELSIF "AzionamentoFesto".AF[#"K_AzionamentoFesto_CMMT-ST"].Input.ExecuteMode AND "AzionamentoFesto".AF[#"K_AzionamentoFesto_CMMT-ST"].Dati.Ready4Motion AND NOT ("AzionamentoFesto".AF[#"K_AzionamentoFesto_CMMT-ST"].Input.ModePos = 4 OR "AzionamentoFesto".AF[#"K_AzionamentoFesto_CMMT-ST"].Input.ModePos = 5 OR "AzionamentoFesto".AF[#"K_AzionamentoFesto_CMMT-ST"].Input.ModePos = 7 OR "AzionamentoFesto".AF[#"K_AzionamentoFesto_CMMT-ST"].Input.ModePos = 8) THEN
       "AzionamentoFesto".AF[#"K_AzionamentoFesto_CMMT-ST"].Dati.ExecuteIntern := TRUE;
       "AzionamentoFesto".AF[#"K_AzionamentoFesto_CMMT-ST"].Dati.ActMode := "AzionamentoFesto".AF[#"K_AzionamentoFesto_CMMT-ST"].Input.ModePos;
       "AzionamentoFesto".AF[#"K_AzionamentoFesto_CMMT-ST"].Dati.StepHome := 0;
   ELSIF "AzionamentoFesto".AF[#"K_AzionamentoFesto_CMMT-ST"].Dati.ExecR_Trig AND ("AzionamentoFesto".AF[#"K_AzionamentoFesto_CMMT-ST"].Input.ModePos = 4 OR "AzionamentoFesto".AF[#"K_AzionamentoFesto_CMMT-ST"].Input.ModePos = 5) THEN
       "AzionamentoFesto".AF[#"K_AzionamentoFesto_CMMT-ST"].Dati.ActMode := "AzionamentoFesto".AF[#"K_AzionamentoFesto_CMMT-ST"].Input.ModePos;
       "AzionamentoFesto".AF[#"K_AzionamentoFesto_CMMT-ST"].Dati.StepHome := 0;
   ELSIF "AzionamentoFesto".AF[#"K_AzionamentoFesto_CMMT-ST"].Input.ExecuteMode AND ("AzionamentoFesto".AF[#"K_AzionamentoFesto_CMMT-ST"].Dati.ActMode = 7 OR "AzionamentoFesto".AF[#"K_AzionamentoFesto_CMMT-ST"].Dati.ActMode = 8) THEN
       "AzionamentoFesto".AF[#"K_AzionamentoFesto_CMMT-ST"].Dati.ExecuteIntern := FALSE;
       "AzionamentoFesto".AF[#"K_AzionamentoFesto_CMMT-ST"].Dati.StepHome := 0;
   ELSIF "AzionamentoFesto".AF[#"K_AzionamentoFesto_CMMT-ST"].Input.ExecuteMode AND "AzionamentoFesto".AF[#"K_AzionamentoFesto_CMMT-ST"].Input.ModePos = 4 THEN

       CASE "AzionamentoFesto".AF[#"K_AzionamentoFesto_CMMT-ST"].Dati.StepHome OF

           0: // homing is active
               IF NOT "AzionamentoFesto".AF[#"K_AzionamentoFesto_CMMT-ST"].Output.AxisRef THEN
                   "AzionamentoFesto".AF[#"K_AzionamentoFesto_CMMT-ST"].Dati.StepHome := 10;
               ELSIF "AzionamentoFesto".AF[#"K_AzionamentoFesto_CMMT-ST"].Output.AxisError OR (NOT "AzionamentoFesto".AF[#"K_AzionamentoFesto_CMMT-ST"].Output.AxisSpFixed AND "AzionamentoFesto".AF[#"K_AzionamentoFesto_CMMT-ST"].Input.ModePos = 4) THEN
                   "AzionamentoFesto".AF[#"K_AzionamentoFesto_CMMT-ST"].Dati.ExecuteIntern := FALSE;
               END_IF;

           10: // wait for homing done
               IF "AzionamentoFesto".AF[#"K_AzionamentoFesto_CMMT-ST"].Output.AxisRef OR "AzionamentoFesto".AF[#"K_AzionamentoFesto_CMMT-ST"].Output.AxisError OR (NOT "AzionamentoFesto".AF[#"K_AzionamentoFesto_CMMT-ST"].Dati.Ready4Motion AND "AzionamentoFesto".AF[#"K_AzionamentoFesto_CMMT-ST"].Input.ModePos = 4) OR "AzionamentoFesto".AF[#"K_AzionamentoFesto_CMMT-ST"].Input.ModePos <> "AzionamentoFesto".AF[#"K_AzionamentoFesto_CMMT-ST"].Dati.ActMode OR NOT "AzionamentoFesto".AF[#"K_AzionamentoFesto_CMMT-ST"].Input.ExecuteMode THEN
                   "AzionamentoFesto".AF[#"K_AzionamentoFesto_CMMT-ST"].Dati.ExecuteIntern := FALSE;
                   "AzionamentoFesto".AF[#"K_AzionamentoFesto_CMMT-ST"].Dati.StepHome := 0;
               END_IF;
       END_CASE;
   ELSIF "AzionamentoFesto".AF[#"K_AzionamentoFesto_CMMT-ST"].Dati.ExecuteIntern AND "AzionamentoFesto".AF[#"K_AzionamentoFesto_CMMT-ST"].Input.ModePos <> "AzionamentoFesto".AF[#"K_AzionamentoFesto_CMMT-ST"].Dati.ActMode THEN
       "AzionamentoFesto".AF[#"K_AzionamentoFesto_CMMT-ST"].Dati.ExecuteIntern := false;
       "AzionamentoFesto".AF[#"K_AzionamentoFesto_CMMT-ST"].Dati.StepHome := 0;
   END_IF;

   //Reset the jog bits if the ModePos has changed
   IF ("AzionamentoFesto".AF[#"K_AzionamentoFesto_CMMT-ST"].Dati.CycWrite.STW1.jog1 OR "AzionamentoFesto".AF[#"K_AzionamentoFesto_CMMT-ST"].Dati.CycWrite.STW1.jog2) AND "AzionamentoFesto".AF[#"K_AzionamentoFesto_CMMT-ST"].Input.ModePos <> "AzionamentoFesto".AF[#"K_AzionamentoFesto_CMMT-ST"].Dati.ActMode THEN
       //Set the jog bits to zero
       "AzionamentoFesto".AF[#"K_AzionamentoFesto_CMMT-ST"].Dati.CycWrite.STW1.jog1 := false;
       "AzionamentoFesto".AF[#"K_AzionamentoFesto_CMMT-ST"].Dati.CycWrite.STW1.jog2 := false;
   END_IF;

   // Positionig mode with relative movement (MDI)
   IF "AzionamentoFesto".AF[#"K_AzionamentoFesto_CMMT-ST"].Input.ModePos = 1 THEN

       // Set the MDI bit
       "AzionamentoFesto".AF[#"K_AzionamentoFesto_CMMT-ST"].Dati.CycWrite.POS_STW1.MDI_Activate := true;

       // positive direction
       "AzionamentoFesto".AF[#"K_AzionamentoFesto_CMMT-ST"].Dati.CycWrite.POS_STW1.PosModulo := "AzionamentoFesto".AF[#"K_AzionamentoFesto_CMMT-ST"].Input.Positive;

       // "festoblockdb".Input.Negative direction
       "AzionamentoFesto".AF[#"K_AzionamentoFesto_CMMT-ST"].Dati.CycWrite.POS_STW1.NegModulo := "AzionamentoFesto".AF[#"K_AzionamentoFesto_CMMT-ST"].Input.Negative;

       // Check if the drive is enabled for a new motion command
       IF "AzionamentoFesto".AF[#"K_AzionamentoFesto_CMMT-ST"].Dati.Ready4Motion THEN

           IF NOT "AzionamentoFesto".AF[#"K_AzionamentoFesto_CMMT-ST"].Dati.CycWrite.STW1.activateTraversing THEN
               "AzionamentoFesto".AF[#"K_AzionamentoFesto_CMMT-ST"].Dati.ExecuteIntern := "AzionamentoFesto".AF[#"K_AzionamentoFesto_CMMT-ST"].Dati.ExecR_Trig;
           END_IF;

           //Start Traversing Task
           "AzionamentoFesto".AF[#"K_AzionamentoFesto_CMMT-ST"].Dati.CycWrite.STW1.activateTraversing := "AzionamentoFesto".AF[#"K_AzionamentoFesto_CMMT-ST"].Dati.ExecuteIntern;

       END_IF;

       // Positionig mode with absolute movement (MDI)
   ELSIF "AzionamentoFesto".AF[#"K_AzionamentoFesto_CMMT-ST"].Input.ModePos = 2 THEN

       // Set the MDI bit
       "AzionamentoFesto".AF[#"K_AzionamentoFesto_CMMT-ST"].Dati.CycWrite.POS_STW1.MDI_Activate := true;

       //set the Absolute bit
       "AzionamentoFesto".AF[#"K_AzionamentoFesto_CMMT-ST"].Dati.CycWrite.POS_STW1.MDI_MOD := true;

       // positive direction
       "AzionamentoFesto".AF[#"K_AzionamentoFesto_CMMT-ST"].Dati.CycWrite.POS_STW1.PosModulo := "AzionamentoFesto".AF[#"K_AzionamentoFesto_CMMT-ST"].Input.Positive;

       // "festoblockdb".Input.Negative direction
       "AzionamentoFesto".AF[#"K_AzionamentoFesto_CMMT-ST"].Dati.CycWrite.POS_STW1.NegModulo := "AzionamentoFesto".AF[#"K_AzionamentoFesto_CMMT-ST"].Input.Negative;

       // Check if the drive is enabled for a new motion command
       IF "AzionamentoFesto".AF[#"K_AzionamentoFesto_CMMT-ST"].Dati.Ready4Motion THEN

           IF NOT "AzionamentoFesto".AF[#"K_AzionamentoFesto_CMMT-ST"].Dati.CycWrite.STW1.activateTraversing THEN
               "AzionamentoFesto".AF[#"K_AzionamentoFesto_CMMT-ST"].Dati.ExecuteIntern := "AzionamentoFesto".AF[#"K_AzionamentoFesto_CMMT-ST"].Dati.ExecR_Trig;
           END_IF;

           //Start Traversing Task
           "AzionamentoFesto".AF[#"K_AzionamentoFesto_CMMT-ST"].Dati.CycWrite.STW1.activateTraversing := "AzionamentoFesto".AF[#"K_AzionamentoFesto_CMMT-ST"].Dati.ExecuteIntern;

       END_IF;

       // Positioning with setup mode for endless motion
   ELSIF "AzionamentoFesto".AF[#"K_AzionamentoFesto_CMMT-ST"].Input.ModePos = 3 THEN
       // Set the MDI bit
       "AzionamentoFesto".AF[#"K_AzionamentoFesto_CMMT-ST"].Dati.CycWrite.POS_STW1.MDI_Activate := true;

       //set the Absolute bit
       "AzionamentoFesto".AF[#"K_AzionamentoFesto_CMMT-ST"].Dati.CycWrite.POS_STW1.MDI_MOD := true;

       //setup mode
       "AzionamentoFesto".AF[#"K_AzionamentoFesto_CMMT-ST"].Dati.CycWrite.POS_STW1.SetupMode := true;

       // positive direction
       "AzionamentoFesto".AF[#"K_AzionamentoFesto_CMMT-ST"].Dati.CycWrite.POS_STW1.PosModulo := "AzionamentoFesto".AF[#"K_AzionamentoFesto_CMMT-ST"].Input.Positive;

       // "festoblockdb".Input.Negative direction
       "AzionamentoFesto".AF[#"K_AzionamentoFesto_CMMT-ST"].Dati.CycWrite.POS_STW1.NegModulo := "AzionamentoFesto".AF[#"K_AzionamentoFesto_CMMT-ST"].Input.Negative;

       // Check if the drive is enabled for a new motion command
       IF "AzionamentoFesto".AF[#"K_AzionamentoFesto_CMMT-ST"].Dati.Ready4Motion THEN

           IF NOT "AzionamentoFesto".AF[#"K_AzionamentoFesto_CMMT-ST"].Dati.CycWrite.STW1.activateTraversing THEN
               "AzionamentoFesto".AF[#"K_AzionamentoFesto_CMMT-ST"].Dati.ExecuteIntern := "AzionamentoFesto".AF[#"K_AzionamentoFesto_CMMT-ST"].Dati.ExecR_Trig;
           END_IF;

           //Start Traversing Task
           "AzionamentoFesto".AF[#"K_AzionamentoFesto_CMMT-ST"].Dati.CycWrite.STW1.activateTraversing := "AzionamentoFesto".AF[#"K_AzionamentoFesto_CMMT-ST"].Dati.ExecuteIntern;

       END_IF;

       //Homing mode done by the drive due to the parametrized homing method
   ELSIF "AzionamentoFesto".AF[#"K_AzionamentoFesto_CMMT-ST"].Input.ModePos = 4 THEN
       // positive direction
       "AzionamentoFesto".AF[#"K_AzionamentoFesto_CMMT-ST"].Dati.CycWrite.POS_STW1.PosModulo := "AzionamentoFesto".AF[#"K_AzionamentoFesto_CMMT-ST"].Input.Positive;

       // "festoblockdb".Input.Negative direction
       "AzionamentoFesto".AF[#"K_AzionamentoFesto_CMMT-ST"].Dati.CycWrite.POS_STW1.NegModulo := "AzionamentoFesto".AF[#"K_AzionamentoFesto_CMMT-ST"].Input.Negative;

       // Check if the drive is enabled for a new motion command
       IF "AzionamentoFesto".AF[#"K_AzionamentoFesto_CMMT-ST"].Dati.Ready4Motion THEN

           //Start homing
           IF NOT "AzionamentoFesto".AF[#"K_AzionamentoFesto_CMMT-ST"].Dati.CycWrite.STW1.StartHoming THEN
               "AzionamentoFesto".AF[#"K_AzionamentoFesto_CMMT-ST"].Dati.ExecuteIntern := "AzionamentoFesto".AF[#"K_AzionamentoFesto_CMMT-ST"].Dati.ExecR_Trig;
           END_IF;

           "AzionamentoFesto".AF[#"K_AzionamentoFesto_CMMT-ST"].Dati.CycWrite.STW1.StartHoming := "AzionamentoFesto".AF[#"K_AzionamentoFesto_CMMT-ST"].Dati.ExecuteIntern;
       END_IF;

       //set the reference point (actual position)
   ELSIF "AzionamentoFesto".AF[#"K_AzionamentoFesto_CMMT-ST"].Input.ModePos = 5 THEN

       // check if there is no error in the drive - this function works also when drive is not enabled
       IF NOT "AzionamentoFesto".AF[#"K_AzionamentoFesto_CMMT-ST"].Output.AxisError THEN

           //Start homing
           IF NOT "AzionamentoFesto".AF[#"K_AzionamentoFesto_CMMT-ST"].Dati.CycWrite.POS_STW2.SetReferencePoint THEN
               "AzionamentoFesto".AF[#"K_AzionamentoFesto_CMMT-ST"].Dati.ExecuteIntern := "AzionamentoFesto".AF[#"K_AzionamentoFesto_CMMT-ST"].Dati.ExecR_Trig;
           END_IF;
           //Set the axis zero point
           "AzionamentoFesto".AF[#"K_AzionamentoFesto_CMMT-ST"].Dati.CycWrite.POS_STW2.SetReferencePoint := "AzionamentoFesto".AF[#"K_AzionamentoFesto_CMMT-ST"].Dati.ExecuteIntern;

       END_IF;

       //Record mode - parametrized records in the drive can be used
   ELSIF "AzionamentoFesto".AF[#"K_AzionamentoFesto_CMMT-ST"].Input.ModePos = 6 THEN

       //set the position number into the record bits 
       IF (DINT_TO_INT("AzionamentoFesto".AF[#"K_AzionamentoFesto_CMMT-ST"].Input.Position) < 0) OR (DINT_TO_INT("AzionamentoFesto".AF[#"K_AzionamentoFesto_CMMT-ST"].Input.Position) > 127) THEN
           // Error, wrong record number
           "AzionamentoFesto".AF[#"K_AzionamentoFesto_CMMT-ST"].Dati.Status := #ERROR_INVALID_TRV_BLOCK;
           "AzionamentoFesto".AF[#"K_AzionamentoFesto_CMMT-ST"].Output.Error := True;
       ELSE
           // error is gone -> set status in operational
           IF "AzionamentoFesto".AF[#"K_AzionamentoFesto_CMMT-ST"].Dati.Status = #ERROR_INVALID_TRV_BLOCK THEN
               "AzionamentoFesto".AF[#"K_AzionamentoFesto_CMMT-ST"].Dati.Status := #STATUS_IN_OPERATION;
               "AzionamentoFesto".AF[#"K_AzionamentoFesto_CMMT-ST"].Output.Error := False;
           END_IF;

           // Record bit 0
           IF (DINT_TO_WORD("AzionamentoFesto".AF[#"K_AzionamentoFesto_CMMT-ST"].Input.Position) AND W#16#01) = W#16#01 THEN
               "AzionamentoFesto".AF[#"K_AzionamentoFesto_CMMT-ST"].Dati.CycWrite.POS_STW1.travBlockBit0 := true;
           END_IF;

           // Record bit 1
           IF (DINT_TO_WORD("AzionamentoFesto".AF[#"K_AzionamentoFesto_CMMT-ST"].Input.Position) AND W#16#02) = W#16#02 THEN
               "AzionamentoFesto".AF[#"K_AzionamentoFesto_CMMT-ST"].Dati.CycWrite.POS_STW1.travBlockBit1 := true;
           END_IF;

           // Record bit 2
           IF (DINT_TO_WORD("AzionamentoFesto".AF[#"K_AzionamentoFesto_CMMT-ST"].Input.Position) AND W#16#04) = W#16#04 THEN
               "AzionamentoFesto".AF[#"K_AzionamentoFesto_CMMT-ST"].Dati.CycWrite.POS_STW1.travBlockBit2 := true;
           END_IF;

           // Record bit 3
           IF (DINT_TO_WORD("AzionamentoFesto".AF[#"K_AzionamentoFesto_CMMT-ST"].Input.Position) AND W#16#08) = W#16#08 THEN
               "AzionamentoFesto".AF[#"K_AzionamentoFesto_CMMT-ST"].Dati.CycWrite.POS_STW1.travBlockBit3 := true;
           END_IF;

           // Record bit 4
           IF (DINT_TO_WORD("AzionamentoFesto".AF[#"K_AzionamentoFesto_CMMT-ST"].Input.Position) AND W#16#10) = W#16#10 THEN
               "AzionamentoFesto".AF[#"K_AzionamentoFesto_CMMT-ST"].Dati.CycWrite.POS_STW1.travBlockBit4 := true;
           END_IF;

           // Record bit 5
           IF (DINT_TO_WORD("AzionamentoFesto".AF[#"K_AzionamentoFesto_CMMT-ST"].Input.Position) AND W#16#20) = W#16#20 THEN
               "AzionamentoFesto".AF[#"K_AzionamentoFesto_CMMT-ST"].Dati.CycWrite.POS_STW1.travBlockBit5 := true;
           END_IF;

           // Record bit 6
           IF (DINT_TO_WORD("AzionamentoFesto".AF[#"K_AzionamentoFesto_CMMT-ST"].Input.Position) AND W#16#40) = W#16#40 THEN
               "AzionamentoFesto".AF[#"K_AzionamentoFesto_CMMT-ST"].Dati.CycWrite.POS_STW1.travBlockBit6 := true;
           END_IF;

           // Check if the drive is enabled for a new motion command
           IF "AzionamentoFesto".AF[#"K_AzionamentoFesto_CMMT-ST"].Dati.Ready4Motion THEN

               IF NOT "AzionamentoFesto".AF[#"K_AzionamentoFesto_CMMT-ST"].Dati.CycWrite.STW1.activateTraversing THEN
                   "AzionamentoFesto".AF[#"K_AzionamentoFesto_CMMT-ST"].Dati.ExecuteIntern := "AzionamentoFesto".AF[#"K_AzionamentoFesto_CMMT-ST"].Dati.ExecR_Trig;
               END_IF;

               //Start Traversing Task
               "AzionamentoFesto".AF[#"K_AzionamentoFesto_CMMT-ST"].Dati.CycWrite.STW1.activateTraversing := "AzionamentoFesto".AF[#"K_AzionamentoFesto_CMMT-ST"].Dati.ExecuteIntern;

           END_IF;
       END_IF;

       //Jog mode - positive or negative
   ELSIF "AzionamentoFesto".AF[#"K_AzionamentoFesto_CMMT-ST"].Input.ModePos = 7 THEN

       // Check if the drive is enabled for a new motion command
       IF "AzionamentoFesto".AF[#"K_AzionamentoFesto_CMMT-ST"].Dati.Ready4Motion THEN

           IF "AzionamentoFesto".AF[#"K_AzionamentoFesto_CMMT-ST"].Dati.Jog1PR_trig AND NOT "AzionamentoFesto".AF[#"K_AzionamentoFesto_CMMT-ST"].Input.Jog2 THEN
               "AzionamentoFesto".AF[#"K_AzionamentoFesto_CMMT-ST"].Dati.CycWrite.STW1.jog1 := TRUE;
               "AzionamentoFesto".AF[#"K_AzionamentoFesto_CMMT-ST"].Dati.ActMode := "AzionamentoFesto".AF[#"K_AzionamentoFesto_CMMT-ST"].Input.ModePos;
           ELSIF NOT "AzionamentoFesto".AF[#"K_AzionamentoFesto_CMMT-ST"].Input.Jog1 THEN
               "AzionamentoFesto".AF[#"K_AzionamentoFesto_CMMT-ST"].Dati.CycWrite.STW1.jog1 := false;
           END_IF;

           IF "AzionamentoFesto".AF[#"K_AzionamentoFesto_CMMT-ST"].Dati.Jog2PR_trig AND NOT "AzionamentoFesto".AF[#"K_AzionamentoFesto_CMMT-ST"].Input.Jog1 THEN
               "AzionamentoFesto".AF[#"K_AzionamentoFesto_CMMT-ST"].Dati.CycWrite.STW1.jog2 := TRUE;
               "AzionamentoFesto".AF[#"K_AzionamentoFesto_CMMT-ST"].Dati.ActMode := "AzionamentoFesto".AF[#"K_AzionamentoFesto_CMMT-ST"].Input.ModePos;
           ELSIF NOT "AzionamentoFesto".AF[#"K_AzionamentoFesto_CMMT-ST"].Input.Jog2 THEN
               "AzionamentoFesto".AF[#"K_AzionamentoFesto_CMMT-ST"].Dati.CycWrite.STW1.jog2 := false;
           END_IF;
       ELSE
           "AzionamentoFesto".AF[#"K_AzionamentoFesto_CMMT-ST"].Dati.CycWrite.STW1.jog1 := false;
           "AzionamentoFesto".AF[#"K_AzionamentoFesto_CMMT-ST"].Dati.CycWrite.STW1.jog2 := false;

       END_IF;

       // jog incremental mode
   ELSIF "AzionamentoFesto".AF[#"K_AzionamentoFesto_CMMT-ST"].Input.ModePos = 8 THEN

       // Check if the drive is enabled for a new motion command
       IF "AzionamentoFesto".AF[#"K_AzionamentoFesto_CMMT-ST"].Dati.Ready4Motion THEN

           //Jog increment
           "AzionamentoFesto".AF[#"K_AzionamentoFesto_CMMT-ST"].Dati.CycWrite.POS_STW2.jog_inc := true;

           IF "AzionamentoFesto".AF[#"K_AzionamentoFesto_CMMT-ST"].Dati.Jog1PMode8R_trig THEN
               "AzionamentoFesto".AF[#"K_AzionamentoFesto_CMMT-ST"].Dati.CycWrite.STW1.jog1 := TRUE;
               "AzionamentoFesto".AF[#"K_AzionamentoFesto_CMMT-ST"].Dati.ActMode := "AzionamentoFesto".AF[#"K_AzionamentoFesto_CMMT-ST"].Input.ModePos;
           ELSIF NOT "AzionamentoFesto".AF[#"K_AzionamentoFesto_CMMT-ST"].Input.Jog1 THEN
               "AzionamentoFesto".AF[#"K_AzionamentoFesto_CMMT-ST"].Dati.CycWrite.STW1.jog1 := false;
           END_IF;

           IF "AzionamentoFesto".AF[#"K_AzionamentoFesto_CMMT-ST"].Dati.Jog2PMode8R_trig THEN
               "AzionamentoFesto".AF[#"K_AzionamentoFesto_CMMT-ST"].Dati.CycWrite.STW1.jog2 := TRUE;
               "AzionamentoFesto".AF[#"K_AzionamentoFesto_CMMT-ST"].Dati.ActMode := "AzionamentoFesto".AF[#"K_AzionamentoFesto_CMMT-ST"].Input.ModePos;
           ELSIF NOT "AzionamentoFesto".AF[#"K_AzionamentoFesto_CMMT-ST"].Input.Jog2 THEN
               "AzionamentoFesto".AF[#"K_AzionamentoFesto_CMMT-ST"].Dati.CycWrite.STW1.jog2 := false;
           END_IF;

           IF "AzionamentoFesto".AF[#"K_AzionamentoFesto_CMMT-ST"].Dati.Jog1PMode8R_trig AND "AzionamentoFesto".AF[#"K_AzionamentoFesto_CMMT-ST"].Dati.Jog2PMode8R_trig THEN
               "AzionamentoFesto".AF[#"K_AzionamentoFesto_CMMT-ST"].Dati.CycWrite.STW1.jog1 := false;
               "AzionamentoFesto".AF[#"K_AzionamentoFesto_CMMT-ST"].Dati.CycWrite.STW1.jog2 := FALSE;
           END_IF;

       ELSE
           "AzionamentoFesto".AF[#"K_AzionamentoFesto_CMMT-ST"].Dati.CycWrite.STW1.jog1 := false;
           "AzionamentoFesto".AF[#"K_AzionamentoFesto_CMMT-ST"].Dati.CycWrite.STW1.jog2 := false;

       END_IF;
   ELSE
       // modepos < 1 or > 8
       "AzionamentoFesto".AF[#"K_AzionamentoFesto_CMMT-ST"].Dati.ExecuteIntern := false;
       "AzionamentoFesto".AF[#"K_AzionamentoFesto_CMMT-ST"].Dati.CycWrite.STW1.activateTraversing := false;
       "AzionamentoFesto".AF[#"K_AzionamentoFesto_CMMT-ST"].Dati.CycWrite.STW1.StartHoming := false;
       "AzionamentoFesto".AF[#"K_AzionamentoFesto_CMMT-ST"].Dati.CycWrite.POS_STW2.SetReferencePoint := false;
       "AzionamentoFesto".AF[#"K_AzionamentoFesto_CMMT-ST"].Dati.StepHome := 0;
       "AzionamentoFesto".AF[#"K_AzionamentoFesto_CMMT-ST"].Dati.statStartCounter := 0;
   END_IF;


   REGION ConfigEPos
       //Maping of the ConfigEPos to the Telegram
       "AzionamentoFesto".AF[#"K_AzionamentoFesto_CMMT-ST"].Dati.CycWrite.STW1.noCoastStop := "AzionamentoFesto".AF[#"K_AzionamentoFesto_CMMT-ST"].Input.ConfigEPos.%X0;         //STW1.1
       "AzionamentoFesto".AF[#"K_AzionamentoFesto_CMMT-ST"].Dati.CycWrite.STW1.noQuickStop := "AzionamentoFesto".AF[#"K_AzionamentoFesto_CMMT-ST"].Input.ConfigEPos.%X1;         //STW1.2
       "AzionamentoFesto".AF[#"K_AzionamentoFesto_CMMT-ST"].Dati.CycWrite.POS_STW2."SW-Limit" := "AzionamentoFesto".AF[#"K_AzionamentoFesto_CMMT-ST"].Input.ConfigEPos.%X2;
       "AzionamentoFesto".AF[#"K_AzionamentoFesto_CMMT-ST"].Dati.CycWrite.POS_STW2."HW-Limit" := "AzionamentoFesto".AF[#"K_AzionamentoFesto_CMMT-ST"].Input.ConfigEPos.%X3;
       "AzionamentoFesto".AF[#"K_AzionamentoFesto_CMMT-ST"].Dati.CycWrite.POS_STW2.ProbeEdgeEval := "AzionamentoFesto".AF[#"K_AzionamentoFesto_CMMT-ST"].Input.ConfigEPos.%X4;
       "AzionamentoFesto".AF[#"K_AzionamentoFesto_CMMT-ST"].Dati.CycWrite.POS_STW2.SelectProbe := "AzionamentoFesto".AF[#"K_AzionamentoFesto_CMMT-ST"].Input.ConfigEPos.%X5;
       "AzionamentoFesto".AF[#"K_AzionamentoFesto_CMMT-ST"].Dati.CycWrite.STW1.ExternalBlockChange := "AzionamentoFesto".AF[#"K_AzionamentoFesto_CMMT-ST"].Input.ConfigEPos.%X6;
       "AzionamentoFesto".AF[#"K_AzionamentoFesto_CMMT-ST"].Dati.CycWrite.POS_STW2.reserved2 := "AzionamentoFesto".AF[#"K_AzionamentoFesto_CMMT-ST"].Input.ConfigEPos.%X7;
       "AzionamentoFesto".AF[#"K_AzionamentoFesto_CMMT-ST"].Dati.CycWrite.POS_STW1.reserved12 := "AzionamentoFesto".AF[#"K_AzionamentoFesto_CMMT-ST"].Input.ConfigEPos.%X8;
       "AzionamentoFesto".AF[#"K_AzionamentoFesto_CMMT-ST"].Dati.CycWrite.STW2.reserved0 := "AzionamentoFesto".AF[#"K_AzionamentoFesto_CMMT-ST"].Input.ConfigEPos.%X9;
       "AzionamentoFesto".AF[#"K_AzionamentoFesto_CMMT-ST"].Dati.CycWrite.STW2.reserved1 := "AzionamentoFesto".AF[#"K_AzionamentoFesto_CMMT-ST"].Input.ConfigEPos.%X10;
       "AzionamentoFesto".AF[#"K_AzionamentoFesto_CMMT-ST"].Dati.CycWrite.STW2.reserved2 := "AzionamentoFesto".AF[#"K_AzionamentoFesto_CMMT-ST"].Input.ConfigEPos.%X11;
       "AzionamentoFesto".AF[#"K_AzionamentoFesto_CMMT-ST"].Dati.CycWrite.STW2.reserved3 := "AzionamentoFesto".AF[#"K_AzionamentoFesto_CMMT-ST"].Input.ConfigEPos.%X12;
       "AzionamentoFesto".AF[#"K_AzionamentoFesto_CMMT-ST"].Dati.CycWrite.STW2.reserved4 := "AzionamentoFesto".AF[#"K_AzionamentoFesto_CMMT-ST"].Input.ConfigEPos.%X13;
       "AzionamentoFesto".AF[#"K_AzionamentoFesto_CMMT-ST"].Dati.CycWrite.STW2.reserved7 := "AzionamentoFesto".AF[#"K_AzionamentoFesto_CMMT-ST"].Input.ConfigEPos.%X14;
       "AzionamentoFesto".AF[#"K_AzionamentoFesto_CMMT-ST"].Dati.CycWrite.STW1.ReleaseBrake := "AzionamentoFesto".AF[#"K_AzionamentoFesto_CMMT-ST"].Input.ReleaseBrake OR "AzionamentoFesto".AF[#"K_AzionamentoFesto_CMMT-ST"].Input.ConfigEPos.%X15;           //STW1.12
       "AzionamentoFesto".AF[#"K_AzionamentoFesto_CMMT-ST"].Dati.CycWrite.STW1.reserved14 := "AzionamentoFesto".AF[#"K_AzionamentoFesto_CMMT-ST"].Input.ConfigEPos.%X16;
       "AzionamentoFesto".AF[#"K_AzionamentoFesto_CMMT-ST"].Dati.CycWrite.STW1.reserved15 := "AzionamentoFesto".AF[#"K_AzionamentoFesto_CMMT-ST"].Input.ConfigEPos.%X17;
       "AzionamentoFesto".AF[#"K_AzionamentoFesto_CMMT-ST"].Dati.CycWrite.POS_STW2.Trackingmode := "AzionamentoFesto".AF[#"K_AzionamentoFesto_CMMT-ST"].Input.ConfigEPos.%X18;    // different mapping to SINA_POS
       "AzionamentoFesto".AF[#"K_AzionamentoFesto_CMMT-ST"].Dati.CycWrite.POS_STW1.reserved7 := "AzionamentoFesto".AF[#"K_AzionamentoFesto_CMMT-ST"].Input.ConfigEPos.%X19;                // reserved
       "AzionamentoFesto".AF[#"K_AzionamentoFesto_CMMT-ST"].Dati.CycWrite.POS_STW1.reserved11 := "AzionamentoFesto".AF[#"K_AzionamentoFesto_CMMT-ST"].Input.ConfigEPos.%X20;               // reserved
       "AzionamentoFesto".AF[#"K_AzionamentoFesto_CMMT-ST"].Dati.CycWrite.POS_STW1.reserved13 := "AzionamentoFesto".AF[#"K_AzionamentoFesto_CMMT-ST"].Input.ConfigEPos.%X21;               // reserved
       "AzionamentoFesto".AF[#"K_AzionamentoFesto_CMMT-ST"].Dati.CycWrite.POS_STW2.reserved13 := "AzionamentoFesto".AF[#"K_AzionamentoFesto_CMMT-ST"].Input.ConfigEPos.%X22;
       "AzionamentoFesto".AF[#"K_AzionamentoFesto_CMMT-ST"].Dati.CycWrite.POS_STW2.reserved4 := "AzionamentoFesto".AF[#"K_AzionamentoFesto_CMMT-ST"].Input.ConfigEPos.%X23;
       "AzionamentoFesto".AF[#"K_AzionamentoFesto_CMMT-ST"].Dati.CycWrite.POS_STW2.reserved6 := "AzionamentoFesto".AF[#"K_AzionamentoFesto_CMMT-ST"].Input.ConfigEPos.%X24;
       "AzionamentoFesto".AF[#"K_AzionamentoFesto_CMMT-ST"].Dati.CycWrite.POS_STW2.reserved7 := "AzionamentoFesto".AF[#"K_AzionamentoFesto_CMMT-ST"].Input.ConfigEPos.%X25;
       "AzionamentoFesto".AF[#"K_AzionamentoFesto_CMMT-ST"].Dati.CycWrite.POS_STW2.reserved12 := "AzionamentoFesto".AF[#"K_AzionamentoFesto_CMMT-ST"].Input.ConfigEPos.%X26;
       "AzionamentoFesto".AF[#"K_AzionamentoFesto_CMMT-ST"].Dati.CycWrite.POS_STW2.reserved13 := "AzionamentoFesto".AF[#"K_AzionamentoFesto_CMMT-ST"].Input.ConfigEPos.%X27;
       "AzionamentoFesto".AF[#"K_AzionamentoFesto_CMMT-ST"].Dati.CycWrite.STW2.reserved5 := "AzionamentoFesto".AF[#"K_AzionamentoFesto_CMMT-ST"].Input.ConfigEPos.%X28;
       "AzionamentoFesto".AF[#"K_AzionamentoFesto_CMMT-ST"].Dati.CycWrite.STW2.reserved6 := "AzionamentoFesto".AF[#"K_AzionamentoFesto_CMMT-ST"].Input.ConfigEPos.%X29;
       "AzionamentoFesto".AF[#"K_AzionamentoFesto_CMMT-ST"].Dati.CycWrite.STW2.TravelToFixStop := "AzionamentoFesto".AF[#"K_AzionamentoFesto_CMMT-ST"].Input.TravelToFixStop OR "AzionamentoFesto".AF[#"K_AzionamentoFesto_CMMT-ST"].Input.ConfigEPos.%X30;     //STW2.8
       "AzionamentoFesto".AF[#"K_AzionamentoFesto_CMMT-ST"].Dati.CycWrite.STW2.reserved9 := "AzionamentoFesto".AF[#"K_AzionamentoFesto_CMMT-ST"].Input.ConfigEPos.%X31;
   END_REGION ;

   REGION Write Output to temp data
       // copy all cyclic data from stat data to tmp buffer
       ////STW1
       #tmpSendBuffer[0].%X0 := "AzionamentoFesto".AF[#"K_AzionamentoFesto_CMMT-ST"].Dati.CycWrite.STW1.on;
       #tmpSendBuffer[0].%X1 := "AzionamentoFesto".AF[#"K_AzionamentoFesto_CMMT-ST"].Dati.CycWrite.STW1.noCoastStop;
       #tmpSendBuffer[0].%X2 := "AzionamentoFesto".AF[#"K_AzionamentoFesto_CMMT-ST"].Dati.CycWrite.STW1.noQuickStop;
       #tmpSendBuffer[0].%X3 := "AzionamentoFesto".AF[#"K_AzionamentoFesto_CMMT-ST"].Dati.CycWrite.STW1.enableOperation;
       #tmpSendBuffer[0].%X4 := "AzionamentoFesto".AF[#"K_AzionamentoFesto_CMMT-ST"].Dati.CycWrite.STW1.cancelTraversing;
       #tmpSendBuffer[0].%X5 := "AzionamentoFesto".AF[#"K_AzionamentoFesto_CMMT-ST"].Dati.CycWrite.STW1.intermediateStop;
       #tmpSendBuffer[0].%X6 := "AzionamentoFesto".AF[#"K_AzionamentoFesto_CMMT-ST"].Dati.CycWrite.STW1.activateTraversing;
       #tmpSendBuffer[0].%X7 := "AzionamentoFesto".AF[#"K_AzionamentoFesto_CMMT-ST"].Dati.CycWrite.STW1.acknowledgeFault;
       #tmpSendBuffer[0].%X8 := "AzionamentoFesto".AF[#"K_AzionamentoFesto_CMMT-ST"].Dati.CycWrite.STW1.jog1;
       #tmpSendBuffer[0].%X9 := "AzionamentoFesto".AF[#"K_AzionamentoFesto_CMMT-ST"].Dati.CycWrite.STW1.jog2;
       #tmpSendBuffer[0].%X10 := "AzionamentoFesto".AF[#"K_AzionamentoFesto_CMMT-ST"].Dati.CycWrite.STW1.controlByPlc;
       #tmpSendBuffer[0].%X11 := "AzionamentoFesto".AF[#"K_AzionamentoFesto_CMMT-ST"].Dati.CycWrite.STW1.StartHoming;
       #tmpSendBuffer[0].%X12 := "AzionamentoFesto".AF[#"K_AzionamentoFesto_CMMT-ST"].Dati.CycWrite.STW1.ReleaseBrake;
       #tmpSendBuffer[0].%X13 := "AzionamentoFesto".AF[#"K_AzionamentoFesto_CMMT-ST"].Dati.CycWrite.STW1.ExternalBlockChange;
       #tmpSendBuffer[0].%X14 := "AzionamentoFesto".AF[#"K_AzionamentoFesto_CMMT-ST"].Dati.CycWrite.STW1.reserved14;
       #tmpSendBuffer[0].%X15 := "AzionamentoFesto".AF[#"K_AzionamentoFesto_CMMT-ST"].Dati.CycWrite.STW1.reserved15;
       //POS_STW1
       #tmpSendBuffer[1].%X0 := "AzionamentoFesto".AF[#"K_AzionamentoFesto_CMMT-ST"].Dati.CycWrite.POS_STW1.travBlockBit0;
       #tmpSendBuffer[1].%X1 := "AzionamentoFesto".AF[#"K_AzionamentoFesto_CMMT-ST"].Dati.CycWrite.POS_STW1.travBlockBit1;
       #tmpSendBuffer[1].%X2 := "AzionamentoFesto".AF[#"K_AzionamentoFesto_CMMT-ST"].Dati.CycWrite.POS_STW1.travBlockBit2;
       #tmpSendBuffer[1].%X3 := "AzionamentoFesto".AF[#"K_AzionamentoFesto_CMMT-ST"].Dati.CycWrite.POS_STW1.travBlockBit3;
       #tmpSendBuffer[1].%X4 := "AzionamentoFesto".AF[#"K_AzionamentoFesto_CMMT-ST"].Dati.CycWrite.POS_STW1.travBlockBit4;
       #tmpSendBuffer[1].%X5 := "AzionamentoFesto".AF[#"K_AzionamentoFesto_CMMT-ST"].Dati.CycWrite.POS_STW1.travBlockBit5;
       #tmpSendBuffer[1].%X6 := "AzionamentoFesto".AF[#"K_AzionamentoFesto_CMMT-ST"].Dati.CycWrite.POS_STW1.travBlockBit6;
       #tmpSendBuffer[1].%X7 := "AzionamentoFesto".AF[#"K_AzionamentoFesto_CMMT-ST"].Dati.CycWrite.POS_STW1.reserved7;
       #tmpSendBuffer[1].%X8 := "AzionamentoFesto".AF[#"K_AzionamentoFesto_CMMT-ST"].Dati.CycWrite.POS_STW1.MDI_MOD;
       #tmpSendBuffer[1].%X9 := "AzionamentoFesto".AF[#"K_AzionamentoFesto_CMMT-ST"].Dati.CycWrite.POS_STW1.PosModulo;
       #tmpSendBuffer[1].%X10 := "AzionamentoFesto".AF[#"K_AzionamentoFesto_CMMT-ST"].Dati.CycWrite.POS_STW1.NegModulo;
       #tmpSendBuffer[1].%X11 := "AzionamentoFesto".AF[#"K_AzionamentoFesto_CMMT-ST"].Dati.CycWrite.POS_STW1.reserved11;
       #tmpSendBuffer[1].%X12 := "AzionamentoFesto".AF[#"K_AzionamentoFesto_CMMT-ST"].Dati.CycWrite.POS_STW1.reserved12;
       #tmpSendBuffer[1].%X13 := "AzionamentoFesto".AF[#"K_AzionamentoFesto_CMMT-ST"].Dati.CycWrite.POS_STW1.reserved13;
       #tmpSendBuffer[1].%X14 := "AzionamentoFesto".AF[#"K_AzionamentoFesto_CMMT-ST"].Dati.CycWrite.POS_STW1.SetupMode;
       #tmpSendBuffer[1].%X15 := "AzionamentoFesto".AF[#"K_AzionamentoFesto_CMMT-ST"].Dati.CycWrite.POS_STW1.MDI_Activate;
       //POS_STW2
       #tmpSendBuffer[2].%X0 := "AzionamentoFesto".AF[#"K_AzionamentoFesto_CMMT-ST"].Dati.CycWrite.POS_STW2.Trackingmode;
       #tmpSendBuffer[2].%X1 := "AzionamentoFesto".AF[#"K_AzionamentoFesto_CMMT-ST"].Dati.CycWrite.POS_STW2.SetReferencePoint;
       #tmpSendBuffer[2].%X2 := "AzionamentoFesto".AF[#"K_AzionamentoFesto_CMMT-ST"].Dati.CycWrite.POS_STW2.reserved2;
       #tmpSendBuffer[2].%X3 := "AzionamentoFesto".AF[#"K_AzionamentoFesto_CMMT-ST"].Dati.CycWrite.POS_STW2.reserved3;
       #tmpSendBuffer[2].%X4 := "AzionamentoFesto".AF[#"K_AzionamentoFesto_CMMT-ST"].Dati.CycWrite.POS_STW2.reserved4;
       #tmpSendBuffer[2].%X5 := "AzionamentoFesto".AF[#"K_AzionamentoFesto_CMMT-ST"].Dati.CycWrite.POS_STW2.jog_inc;
       #tmpSendBuffer[2].%X6 := "AzionamentoFesto".AF[#"K_AzionamentoFesto_CMMT-ST"].Dati.CycWrite.POS_STW2.reserved6;
       #tmpSendBuffer[2].%X7 := "AzionamentoFesto".AF[#"K_AzionamentoFesto_CMMT-ST"].Dati.CycWrite.POS_STW2.reserved7;
       #tmpSendBuffer[2].%X8 := "AzionamentoFesto".AF[#"K_AzionamentoFesto_CMMT-ST"].Dati.CycWrite.POS_STW2.FlyingRef;
       #tmpSendBuffer[2].%X9 := "AzionamentoFesto".AF[#"K_AzionamentoFesto_CMMT-ST"].Dati.CycWrite.POS_STW2.reserved9;
       #tmpSendBuffer[2].%X10 := "AzionamentoFesto".AF[#"K_AzionamentoFesto_CMMT-ST"].Dati.CycWrite.POS_STW2.SelectProbe;
       #tmpSendBuffer[2].%X11 := "AzionamentoFesto".AF[#"K_AzionamentoFesto_CMMT-ST"].Dati.CycWrite.POS_STW2.ProbeEdgeEval;
       #tmpSendBuffer[2].%X12 := "AzionamentoFesto".AF[#"K_AzionamentoFesto_CMMT-ST"].Dati.CycWrite.POS_STW2.reserved12;
       #tmpSendBuffer[2].%X13 := "AzionamentoFesto".AF[#"K_AzionamentoFesto_CMMT-ST"].Dati.CycWrite.POS_STW2.reserved13;
       #tmpSendBuffer[2].%X14 := "AzionamentoFesto".AF[#"K_AzionamentoFesto_CMMT-ST"].Dati.CycWrite.POS_STW2."SW-Limit";
       #tmpSendBuffer[2].%X15 := "AzionamentoFesto".AF[#"K_AzionamentoFesto_CMMT-ST"].Dati.CycWrite.POS_STW2."HW-Limit";
       //STW2
       #tmpSendBuffer[3].%X0 := "AzionamentoFesto".AF[#"K_AzionamentoFesto_CMMT-ST"].Dati.CycWrite.STW2.reserved0;
       #tmpSendBuffer[3].%X1 := "AzionamentoFesto".AF[#"K_AzionamentoFesto_CMMT-ST"].Dati.CycWrite.STW2.reserved1;
       #tmpSendBuffer[3].%X2 := "AzionamentoFesto".AF[#"K_AzionamentoFesto_CMMT-ST"].Dati.CycWrite.STW2.reserved2;
       #tmpSendBuffer[3].%X3 := "AzionamentoFesto".AF[#"K_AzionamentoFesto_CMMT-ST"].Dati.CycWrite.STW2.reserved3;
       #tmpSendBuffer[3].%X4 := "AzionamentoFesto".AF[#"K_AzionamentoFesto_CMMT-ST"].Dati.CycWrite.STW2.reserved4;
       #tmpSendBuffer[3].%X5 := "AzionamentoFesto".AF[#"K_AzionamentoFesto_CMMT-ST"].Dati.CycWrite.STW2.reserved5;
       #tmpSendBuffer[3].%X6 := "AzionamentoFesto".AF[#"K_AzionamentoFesto_CMMT-ST"].Dati.CycWrite.STW2.reserved6;
       #tmpSendBuffer[3].%X7 := "AzionamentoFesto".AF[#"K_AzionamentoFesto_CMMT-ST"].Dati.CycWrite.STW2.reserved7;
       #tmpSendBuffer[3].%X8 := "AzionamentoFesto".AF[#"K_AzionamentoFesto_CMMT-ST"].Dati.CycWrite.STW2.TravelToFixStop;
       #tmpSendBuffer[3].%X9 := "AzionamentoFesto".AF[#"K_AzionamentoFesto_CMMT-ST"].Dati.CycWrite.STW2.reserved9;
       #tmpSendBuffer[3].%X10 := "AzionamentoFesto".AF[#"K_AzionamentoFesto_CMMT-ST"].Dati.CycWrite.STW2.reserved10;
       #tmpSendBuffer[3].%X11 := "AzionamentoFesto".AF[#"K_AzionamentoFesto_CMMT-ST"].Dati.CycWrite.STW2.reserved11;
       #tmpSendBuffer[3].%X12 := "AzionamentoFesto".AF[#"K_AzionamentoFesto_CMMT-ST"].Dati.CycWrite.STW2.signOfLifeBit0;
       #tmpSendBuffer[3].%X13 := "AzionamentoFesto".AF[#"K_AzionamentoFesto_CMMT-ST"].Dati.CycWrite.STW2.signOfLifeBit1;
       #tmpSendBuffer[3].%X14 := "AzionamentoFesto".AF[#"K_AzionamentoFesto_CMMT-ST"].Dati.CycWrite.STW2.signOfLifeBit2;
       #tmpSendBuffer[3].%X15 := "AzionamentoFesto".AF[#"K_AzionamentoFesto_CMMT-ST"].Dati.CycWrite.STW2.signOfLifeBit3;

       //Override
       #tmpSendBuffer[4] := "AzionamentoFesto".AF[#"K_AzionamentoFesto_CMMT-ST"].Dati.CycWrite.Override;

       //TargetPos
       #tempDWord := DINT_TO_DWORD("AzionamentoFesto".AF[#"K_AzionamentoFesto_CMMT-ST"].Dati.CycWrite.MDI_TARPOS);
       #tmpSendBuffer[5] := #tempDWord.%W1;
       #tmpSendBuffer[6] := #tempDWord.%W0;

       //TargetVelocity
       #tempDWord := DINT_TO_DWORD("AzionamentoFesto".AF[#"K_AzionamentoFesto_CMMT-ST"].Dati.CycWrite.MDI_VELOCITY);
       #tmpSendBuffer[7] := #tempDWord.%W1;
       #tmpSendBuffer[8] := #tempDWord.%W0;

       // ACC, DEC
       #tmpSendBuffer[9] := "AzionamentoFesto".AF[#"K_AzionamentoFesto_CMMT-ST"].Dati.CycWrite.MDI_ACC;
       #tmpSendBuffer[10] := "AzionamentoFesto".AF[#"K_AzionamentoFesto_CMMT-ST"].Dati.CycWrite.MDI_DEC;
       #tmpSendBuffer[11] := "AzionamentoFesto".AF[#"K_AzionamentoFesto_CMMT-ST"].Dati.CycWrite.reserved11;
   END_REGION ;

   REGION Write Cyclic Data of Telegramm 111
       // Write cyclic telegram 111
       "AzionamentoFesto".AF[#"K_AzionamentoFesto_CMMT-ST"].Dati.RetDPWR := DPWR_DAT(LADDR := "AzionamentoFesto".AF[#"K_AzionamentoFesto_CMMT-ST"].Input.HardwareId,
                                                                                     RECORD := #tmpSendBuffer);

       // write SETIO status to diagId
       IF "AzionamentoFesto".AF[#"K_AzionamentoFesto_CMMT-ST"].Dati.RetDPWR <> 0 THEN
           "AzionamentoFesto".AF[#"K_AzionamentoFesto_CMMT-ST"].Output.Error := true;
           "AzionamentoFesto".AF[#"K_AzionamentoFesto_CMMT-ST"].Dati.Status := #ERROR_DPWR_DAT;
           "AzionamentoFesto".AF[#"K_AzionamentoFesto_CMMT-ST"].Output.DiagID := INT_TO_WORD("AzionamentoFesto".AF[#"K_AzionamentoFesto_CMMT-ST"].Dati.RetDPWR);
       ELSE
           // set the Diag status back "in operation"
           IF "AzionamentoFesto".AF[#"K_AzionamentoFesto_CMMT-ST"].Dati.Status = #ERROR_DPWR_DAT THEN
               "AzionamentoFesto".AF[#"K_AzionamentoFesto_CMMT-ST"].Dati.Status := #STATUS_IN_OPERATION;
               "AzionamentoFesto".AF[#"K_AzionamentoFesto_CMMT-ST"].Output.DiagID := 0;
               "AzionamentoFesto".AF[#"K_AzionamentoFesto_CMMT-ST"].Output.Error := False;
           END_IF;

       END_IF;
       //Set the Status Output
       "AzionamentoFesto".AF[#"K_AzionamentoFesto_CMMT-ST"].Output.Status := "AzionamentoFesto".AF[#"K_AzionamentoFesto_CMMT-ST"].Dati.Status;
       "AzionamentoFesto".AF[#"K_AzionamentoFesto_CMMT-ST"].Output.ActMode := "AzionamentoFesto".AF[#"K_AzionamentoFesto_CMMT-ST"].Dati.ActMode;
   END_REGION
END_REGION
END_FUNCTION
